SPLINE
SPL {X  -162.820, Y  +621.304, Z    +0.000, E1   +22.259, E3 +549839.256}
SPL {X  -162.820, Y  +618.758, Z    +0.000, E1   +22.239, E3 +549852.407}
SPL {X  -162.820, Y  +616.062, Z    +0.000, E1   +22.275, E3 +549865.828}
SPL {X  -162.820, Y  +613.536, Z    +0.000, E1   +22.242, E3 +549878.949}
SPL {X  -162.820, Y  +611.128, Z    +0.000, E1   +22.252, E3 +549891.120}
SPL {X  -162.820, Y  +608.428, Z    +0.000, E1   +22.255, E3 +549904.904}
SPL {X  -162.820, Y  +605.178, Z    +0.000, E1   +22.267, E3 +549921.436}
SPL {X  -162.820, Y  +602.350, Z    +0.000, E1   +22.224, E3 +549936.053}
SPL {X  -162.820, Y  +599.842, Z    +0.000, E1   +22.298, E3 +549948.204}
SPL {X  -162.820, Y  +597.194, Z    +0.000, E1   +22.253, E3 +549962.125}
SPL {X  -162.820, Y  +594.779, Z    +0.000, E1   +22.284, E3 +549974.029}
SPL {X  -162.820, Y  +592.389, Z    +0.000, E1   +22.245, E3 +549986.646}
SPL {X  -162.820, Y  +589.492, Z    +0.000, E1   +22.304, E3 +550000.830}
SPL {X  -162.820, Y  +587.447, Z    +0.000, E1   +22.279, E3 +550011.359}
SPL {X  -162.820, Y  +585.192, Z    +0.000, E1   +22.298, E3 +550022.769}
SPL {X  -162.820, Y  +582.610, Z    +0.000, E1   +22.234, E3 +550036.393}
SPL {X  -162.820, Y  +580.317, Z    +0.000, E1   +22.300, E3 +550047.447}
SPL {X  -162.820, Y  +578.878, Z    +0.000, E1   +22.272, E3 +550054.956}
SPL {X  -162.820, Y  +576.856, Z    +0.000, E1   +22.233, E3 +550065.715}
SPL {X  -162.820, Y  +574.811, Z    +0.000, E1   +22.236, E3 +550075.978}
SPL {X  -162.820, Y  +572.645, Z    +0.000, E1   +22.246, E3 +550087.074}
SPL {X  -162.820, Y  +569.475, Z    +0.000, E1   +22.269, E3 +550103.080}
SPL {X  -162.820, Y  +565.838, Z    +0.000, E1   +22.271, E3 +550121.675}
SPL {X  -162.820, Y  +562.162, Z    +0.000, E1   +22.252, E3 +550140.492}
SPL {X  -162.820, Y  +558.919, Z    +0.000, E1   +22.286, E3 +550156.655}
SPL {X  -162.820, Y  +556.169, Z    +0.000, E1   +22.295, E3 +550170.484}
SPL {X  -162.820, Y  +553.294, Z    +0.000, E1   +22.266, E3 +550185.482}
SPL {X  -162.820, Y  +550.136, Z    +0.000, E1   +22.258, E3 +550201.595}
SPL {X  -162.820, Y  +546.694, Z    +0.000, E1   +22.290, E3 +550218.917}
SPL {X  -162.820, Y  +543.558, Z    +0.000, E1   +22.285, E3 +550234.780}
SPL {X  -162.820, Y  +541.633, Z    +0.000, E1   +22.257, E3 +550244.708}
SPL {X  -162.820, Y  +539.116, Z    +0.000, E1   +22.302, E3 +550257.319}
SPL {X  -162.820, Y  +536.913, Z    +0.000, E1   +22.192, E3 +550269.243}
SPL {X  -162.820, Y  +534.880, Z    +0.000, E1   +22.252, E3 +550279.197}
SPL {X  -162.820, Y  +532.896, Z    +0.000, E1   +22.234, E3 +550289.357}
SPL {X  -162.820, Y  +531.056, Z    +0.000, E1   +22.251, E3 +550298.639}
SPL {X  -162.820, Y  +528.708, Z    +0.000, E1   +22.319, E3 +550310.021}
SPL {X  -162.820, Y  +525.932, Z    +0.000, E1   +22.258, E3 +550324.777}
SPL {X  -162.820, Y  +522.524, Z    +0.000, E1   +22.326, E3 +550341.501}
SPL {X  -162.820, Y  +519.457, Z    +0.000, E1   +22.481, E3 +550355.630}
SPL {X  -162.820, Y  +506.285, Z    +0.000, E1   +28.538, E3 +550367.088}
SPL {X  -162.820, Y  +504.441, Z    +0.000, E1   +27.574, E3 +550381.430}
SPL {X  -162.820, Y  +503.215, Z    +0.000, E1   +26.369, E3 +550394.937}
SPL {X  -162.820, Y  +502.265, Z    +0.000, E1   +25.287, E3 +550407.419}
SPL {X  -162.820, Y  +501.060, Z    +0.000, E1   +24.081, E3 +550422.160}
SPL {X  -162.820, Y  +500.336, Z    +0.000, E1   +23.110, E3 +550433.299}
SPL {X  -162.820, Y  +499.240, Z    +0.000, E1   +22.316, E3 +550445.610}
SPL {X  -162.820, Y  +498.027, Z    +0.000, E1   +21.516, E3 +550458.518}
SPL {X  -162.820, Y  +495.897, Z    +0.000, E1   +21.662, E3 +550468.438}
SPL {X  -162.820, Y  +493.717, Z    +0.000, E1   +21.704, E3 +550479.544}
SPL {X  -162.820, Y  +491.396, Z    +0.000, E1   +21.707, E3 +550491.668}
SPL {X  -162.820, Y  +488.560, Z    +0.000, E1   +21.695, E3 +550506.778}
SPL {X  -162.820, Y  +485.661, Z    +0.000, E1   +21.712, E3 +550521.663}
SPL {X  -162.820, Y  +483.668, Z    +0.000, E1   +21.664, E3 +550532.491}
SPL {X  -162.820, Y  +481.739, Z    +0.000, E1   +21.704, E3 +550542.204}
SPL {X  -162.820, Y  +479.894, Z    +0.000, E1   +21.695, E3 +550551.992}
SPL {X  -162.820, Y  +477.685, Z    +0.000, E1   +21.656, E3 +550563.929}
SPL {X  -162.820, Y  +475.419, Z    +0.000, E1   +21.711, E3 +550575.282}
SPL {X  -162.820, Y  +473.301, Z    +0.000, E1   +21.712, E3 +550586.379}
SPL {X  -162.820, Y  +470.965, Z    +0.000, E1   +21.700, E3 +550598.724}
SPL {X  -162.820, Y  +469.036, Z    +0.000, E1   +21.695, E3 +550608.768}
SPL {X  -162.820, Y  +467.138, Z    +0.000, E1   +21.678, E3 +550618.939}
SPL {X  -162.820, Y  +465.011, Z    +0.000, E1   +21.692, E3 +550629.922}
SPL {X  -162.820, Y  +462.669, Z    +0.000, E1   +21.752, E3 +550641.702}
SPL {X  -162.820, Y  +460.725, Z    +0.000, E1   +21.689, E3 +550652.315}
SPL {X  -162.820, Y  +458.666, Z    +0.000, E1   +21.695, E3 +550663.127}
SPL {X  -162.820, Y  +456.431, Z    +0.000, E1   +21.708, E3 +550674.656}
SPL {X  -162.820, Y  +454.628, Z    +0.000, E1   +21.674, E3 +550684.374}
SPL {X  -162.820, Y  +452.690, Z    +0.000, E1   +21.773, E3 +550693.648}
SPL {X  -162.820, Y  +450.610, Z    +0.000, E1   +21.698, E3 +550705.247}
SPL {X  -162.820, Y  +448.170, Z    +0.000, E1   +21.667, E3 +550718.268}
SPL {X  -162.820, Y  +446.246, Z    +0.000, E1   +21.696, E3 +550728.086}
SPL {X  -162.820, Y  +443.784, Z    +0.000, E1   +21.713, E3 +550740.872}
SPL {X  -162.820, Y  +441.754, Z    +0.000, E1   +21.708, E3 +550751.424}
SPL {X  -162.820, Y  +439.933, Z    +0.000, E1   +21.690, E3 +550761.188}
SPL {X  -162.820, Y  +437.628, Z    +0.000, E1   +21.678, E3 +550773.376}
SPL {X  -162.820, Y  +435.262, Z    +0.000, E1   +21.727, E3 +550785.311}
SPL {X  -162.820, Y  +433.510, Z    +0.000, E1   +21.692, E3 +550794.725}
SPL {X  -162.820, Y  +431.492, Z    +0.000, E1   +21.686, E3 +550805.421}
SPL {X  -162.820, Y  +429.074, Z    +0.000, E1   +21.710, E3 +550817.873}
SPL {X  -162.820, Y  +427.020, Z    +0.000, E1   +21.674, E3 +550828.874}
SPL {X  -162.820, Y  +425.215, Z    +0.000, E1   +21.693, E3 +550838.177}
SPL {X  -162.820, Y  +422.986, Z    +0.000, E1   +21.685, E3 +550849.988}
SPL {X  -162.820, Y  +420.528, Z    +0.000, E1   +21.706, E3 +550862.638}
SPL {X  -162.820, Y  +418.116, Z    +0.000, E1   +21.761, E3 +550874.785}
SPL {X  -162.820, Y  +416.127, Z    +0.000, E1   +21.715, E3 +550885.490}
SPL {X  -162.820, Y  +414.361, Z    +0.000, E1   +21.613, E3 +550895.678}
SPL {X  -162.820, Y  +411.450, Z    +0.000, E1   +21.710, E3 +550910.251}
SPL {X  -162.820, Y  +408.590, Z    +0.000, E1   +21.735, E3 +550924.877}
SPL {X  -162.820, Y  +406.238, Z    +0.000, E1   +21.697, E3 +550937.526}
SPL {X  -162.820, Y  +404.001, Z    +0.000, E1   +21.723, E3 +550948.955}
SPL {X  -162.820, Y  +402.223, Z    +0.000, E1   +21.697, E3 +550958.440}
SPL {X  -162.820, Y  +400.348, Z    +0.000, E1   +21.713, E3 +550968.166}
SPL {X  -162.820, Y  +398.298, Z    +0.000, E1   +21.721, E3 +550978.782}
SPL {X  -162.820, Y  +396.371, Z    +0.000, E1   +21.713, E3 +550988.964}
SPL {X  -162.820, Y  +394.508, Z    +0.000, E1   +21.616, E3 +550999.519}
SPL {X  -162.820, Y  +392.435, Z    +0.000, E1   +21.681, E3 +551009.873}
SPL {X  -162.820, Y  +389.390, Z    +0.000, E1   +21.742, E3 +551025.479}
SPL {X  -162.820, Y  +386.818, Z    +0.000, E1   +21.679, E3 +551039.238}
SPL {X  -162.820, Y  +384.697, Z    +0.000, E1   +21.693, E3 +551050.308}
SPL {X  -162.820, Y  +382.288, Z    +0.000, E1   +21.742, E3 +551062.432}
SPL {X  -162.820, Y  +380.381, Z    +0.000, E1   +21.655, E3 +551073.157}
SPL {X  -162.808, Y  +378.512, Z    +0.000, E1   +21.736, E3 +551082.209}
SPL {X  -162.776, Y  +376.710, Z    +0.000, E1   +21.698, E3 +551092.008}
SPL {X  -162.707, Y  +374.438, Z    +0.000, E1   +21.688, E3 +551104.012}
SPL {X  -162.607, Y  +372.171, Z    +0.000, E1   +21.692, E3 +551115.812}
SPL {X  -162.494, Y  +370.197, Z    +0.000, E1   +21.655, E3 +551126.438}
SPL {X  -162.349, Y  +368.131, Z    +0.000, E1   +21.624, E3 +551137.556}
SPL {X  -162.161, Y  +365.866, Z    +0.000, E1   +21.642, E3 +551149.241}
SPL {X  -161.927, Y  +363.466, Z    +0.000, E1   +21.730, E3 +551161.013}
SPL {X  -160.290, Y  +351.907, Z    +0.000, E1   +27.562, E3 +551168.591}
SPL {X  -159.725, Y  +348.905, Z    +0.000, E1   +26.136, E3 +551193.826}
ENDSPLINE

SPLINE
SPL {X  -160.871, Y  +355.385, Z    +0.000, E1   +21.841, E3 +551202.669}
SPL {X  -161.833, Y  +362.603, Z    +0.000, E1   +17.021, E3 +551212.700}
ENDSPLINE

SPLINE
SPL {X  -160.786, Y  +354.842, Z    +0.000, E1   +19.274, E3 +551244.855}
ENDSPLINE

SPLINE
SPL {X  -162.485, Y  +370.062, Z    +0.000, E1   +10.606, E3 +551251.233}
SPL {X  -162.818, Y  +379.636, Z    +0.000, E1    +5.115, E3 +551240.582}
SPL {X  -162.820, Y  +386.976, Z    +0.000, E1    +0.144, E3 +551239.681}
SPL {X  -162.820, Y  +391.982, Z    +0.000, E1    -3.443, E3 +551246.446}
SPL {X  -162.820, Y  +399.630, Z    +0.000, E1    -9.426, E3 +551248.954}
SPL {X  -162.820, Y  +408.127, Z    +0.000, E1   -18.417, E3 +551235.242}
SPL {X  -162.820, Y  +420.083, Z    +0.000, E1   -24.325, E3 +551255.718}
SPL {X  -162.820, Y  +428.527, Z    +0.000, E1   -26.988, E3 +551273.010}
SPL {X  -162.820, Y  +431.191, Z    +0.000, E1   -23.548, E3 +551307.863}
SPL {X  -162.820, Y  +432.946, Z    +0.000, E1   -22.795, E3 +551322.266}
SPL {X  -162.820, Y  +434.888, Z    +0.000, E1   -22.823, E3 +551331.673}
SPL {X  -162.820, Y  +436.834, Z    +0.000, E1   -22.779, E3 +551341.633}
SPL {X  -162.820, Y  +438.868, Z    +0.000, E1   -22.837, E3 +551351.287}
SPL {X  -162.820, Y  +441.351, Z    +0.000, E1   -22.805, E3 +551363.862}
SPL {X  -162.820, Y  +443.809, Z    +0.000, E1   -22.804, E3 +551376.028}
SPL {X  -162.820, Y  +446.105, Z    +0.000, E1   -22.815, E3 +551387.270}
SPL {X  -162.820, Y  +447.974, Z    +0.000, E1   -22.856, E3 +551396.173}
SPL {X  -162.820, Y  +449.911, Z    +0.000, E1   -22.774, E3 +551406.448}
SPL {X  -162.820, Y  +451.861, Z    +0.000, E1   -22.750, E3 +551416.295}
SPL {X  -162.820, Y  +454.167, Z    +0.000, E1   -22.842, E3 +551427.025}
SPL {X  -162.820, Y  +456.529, Z    +0.000, E1   -22.855, E3 +551438.553}
SPL {X  -162.820, Y  +458.725, Z    +0.000, E1   -22.793, E3 +551449.958}
SPL {X  -162.820, Y  +461.700, Z    +0.000, E1   -22.822, E3 +551464.580}
SPL {X  -162.820, Y  +464.633, Z    +0.000, E1   -22.813, E3 +551479.077}
SPL {X  -162.820, Y  +466.699, Z    +0.000, E1   -22.824, E3 +551489.123}
SPL {X  -162.820, Y  +468.655, Z    +0.000, E1   -22.858, E3 +551498.567}
SPL {X  -162.820, Y  +470.892, Z    +0.000, E1   -22.837, E3 +551509.805}
SPL {X  -162.820, Y  +472.726, Z    +0.000, E1   -22.777, E3 +551519.344}
SPL {X  -162.820, Y  +475.118, Z    +0.000, E1   -22.777, E3 +551531.316}
SPL {X  -162.820, Y  +478.177, Z    +0.000, E1   -22.834, E3 +551546.008}
SPL {X  -162.820, Y  +481.034, Z    +0.000, E1   -22.831, E3 +551560.146}
SPL {X  -162.820, Y  +483.391, Z    +0.000, E1   -22.793, E3 +551572.082}
SPL {X  -162.820, Y  +486.307, Z    +0.000, E1   -22.833, E3 +551586.336}
SPL {X  -162.820, Y  +488.828, Z    +0.000, E1   -22.793, E3 +551598.979}
SPL {X  -162.820, Y  +491.768, Z    +0.000, E1   -22.852, E3 +551613.276}
SPL {X  -162.820, Y  +495.526, Z    +0.000, E1   -22.833, E3 +551632.047}
SPL {X  -162.820, Y  +499.330, Z    +0.000, E1   -22.841, E3 +551650.828}
SPL {X  -162.820, Y  +503.049, Z    +0.000, E1   -22.823, E3 +551669.377}
SPL {X  -162.820, Y  +506.908, Z    +0.000, E1   -22.877, E3 +551688.047}
SPL {X  -162.820, Y  +510.068, Z    +0.000, E1   -22.761, E3 +551704.519}
SPL {X  -162.820, Y  +512.359, Z    +0.000, E1   -22.823, E3 +551715.250}
SPL {X  -162.820, Y  +513.873, Z    +0.000, E1   -22.800, E3 +551722.937}
SPL {X  -162.820, Y  +516.100, Z    +0.000, E1   -22.809, E3 +551734.014}
SPL {X  -162.820, Y  +518.662, Z    +0.000, E1   -22.847, E3 +551746.312}
SPL {X  -162.820, Y  +520.641, Z    +0.000, E1   -22.790, E3 +551756.553}
SPL {X  -162.820, Y  +523.535, Z    +0.000, E1   -22.857, E3 +551770.522}
SPL {X  -162.820, Y  +526.661, Z    +0.000, E1   -22.801, E3 +551786.346}
SPL {X  -162.820, Y  +528.725, Z    +0.000, E1   -22.770, E3 +551796.715}
SPL {X  -162.820, Y  +530.303, Z    +0.000, E1   -22.798, E3 +551804.335}
SPL {X  -162.820, Y  +532.614, Z    +0.000, E1   -22.828, E3 +551815.603}
SPL {X  -162.820, Y  +534.838, Z    +0.000, E1   -22.864, E3 +551826.232}
SPL {X  -162.820, Y  +536.882, Z    +0.000, E1   -22.782, E3 +551837.087}
SPL {X  -162.820, Y  +539.194, Z    +0.000, E1   -22.826, E3 +551848.135}
SPL {X  -162.820, Y  +541.555, Z    +0.000, E1   -22.817, E3 +551859.950}
SPL {X  -162.820, Y  +543.728, Z    +0.000, E1   -22.799, E3 +551870.807}
SPL {X  -162.820, Y  +545.925, Z    +0.000, E1   -22.803, E3 +551881.677}
SPL {X  -162.820, Y  +549.071, Z    +0.000, E1   -22.836, E3 +551897.205}
SPL {X  -162.820, Y  +553.089, Z    +0.000, E1   -22.838, E3 +551917.105}
SPL {X  -162.820, Y  +556.430, Z    +0.000, E1   -22.821, E3 +551933.606}
SPL {X  -162.820, Y  +558.974, Z    +0.000, E1   -22.806, E3 +551946.306}
SPL {X  -162.820, Y  +562.171, Z    +0.000, E1   -22.845, E3 +551962.004}
SPL {X  -162.820, Y  +565.170, Z    +0.000, E1   -22.801, E3 +551977.017}
SPL {X  -162.820, Y  +567.308, Z    +0.000, E1   -22.750, E3 +551988.033}
SPL {X  -162.820, Y  +570.378, Z    +0.000, E1   -22.843, E3 +552002.657}
SPL {X  -162.820, Y  +573.634, Z    +0.000, E1   -22.827, E3 +552018.801}
SPL {X  -162.820, Y  +576.228, Z    +0.000, E1   -22.814, E3 +552031.697}
SPL {X  -162.820, Y  +578.553, Z    +0.000, E1   -22.801, E3 +552043.313}
SPL {X  -162.820, Y  +581.064, Z    +0.000, E1   -22.823, E3 +552055.597}
SPL {X  -162.820, Y  +583.435, Z    +0.000, E1   -22.808, E3 +552067.419}
SPL {X  -162.820, Y  +585.410, Z    +0.000, E1   -22.764, E3 +552077.555}
SPL {X  -162.820, Y  +587.676, Z    +0.000, E1   -22.853, E3 +552088.069}
SPL {X  -162.820, Y  +590.707, Z    +0.000, E1   -22.855, E3 +552103.220}
SPL {X  -162.820, Y  +593.650, Z    +0.000, E1   -22.810, E3 +552117.980}
SPL {X  -162.820, Y  +595.830, Z    +0.000, E1   -22.828, E3 +552128.596}
SPL {X  -162.820, Y  +598.094, Z    +0.000, E1   -22.843, E3 +552139.709}
SPL {X  -162.820, Y  +600.420, Z    +0.000, E1   -22.826, E3 +552151.340}
SPL {X  -162.820, Y  +602.573, Z    +0.000, E1   -22.830, E3 +552161.925}
SPL {X  -162.820, Y  +604.828, Z    +0.000, E1   -22.784, E3 +552173.564}
SPL {X  -162.820, Y  +608.133, Z    +0.000, E1   -22.831, E3 +552189.682}
SPL {X  -162.820, Y  +611.103, Z    +0.000, E1   -22.785, E3 +552204.607}
SPL {X  -162.820, Y  +613.294, Z    +0.000, E1   -22.780, E3 +552215.480}
SPL {X  -162.820, Y  +615.356, Z    +0.000, E1   -22.799, E3 +552225.538}
SPL {X  -162.820, Y  +617.439, Z    +0.000, E1   -22.808, E3 +552235.796}
SPL {X  -162.820, Y  +619.665, Z    +0.000, E1   -22.817, E3 +552246.764}
SPL {X  -162.820, Y  +621.733, Z    +0.000, E1   -22.759, E3 +552257.488}
SPL {X  -162.820, Y  +624.076, Z    +0.000, E1   -22.774, E3 +552268.993}
SPL {X  -162.820, Y  +627.244, Z    +0.000, E1   -22.803, E3 +552284.675}
SPL {X  -162.820, Y  +630.349, Z    +0.000, E1   -22.766, E3 +552300.207}
SPL {X  -162.820, Y  +632.572, Z    +0.000, E1   -22.785, E3 +552311.014}
SPL {X  -162.820, Y  +634.507, Z    +0.000, E1   -22.784, E3 +552320.653}
SPL {X  -162.820, Y  +636.863, Z    +0.000, E1   -22.760, E3 +552332.575}
SPL {X  -162.820, Y  +640.111, Z    +0.000, E1   -22.809, E3 +552348.458}
SPL {X  -162.820, Y  +643.449, Z    +0.000, E1   -22.796, E3 +552364.975}
SPL {X  -162.820, Y  +645.630, Z    +0.000, E1   -22.795, E3 +552375.671}
SPL {X  -162.820, Y  +647.561, Z    +0.000, E1   -22.705, E3 +552386.122}
SPL {X  -162.820, Y  +651.051, Z    +0.000, E1   -22.833, E3 +552402.542}
SPL {X  -162.820, Y  +653.898, Z    +0.000, E1   -22.796, E3 +552416.727}
SPL {X  -162.820, Y  +656.161, Z    +0.000, E1   -22.812, E3 +552427.849}
SPL {X  -162.820, Y  +658.384, Z    +0.000, E1   -22.822, E3 +552438.715}
SPL {X  -162.820, Y  +660.215, Z    +0.000, E1   -22.649, E3 +552449.306}
SPL {X  -162.820, Y  +662.823, Z    +0.000, E1   -22.799, E3 +552461.014}
SPL {X  -162.820, Y  +665.862, Z    +0.000, E1   -22.864, E3 +552475.713}
SPL {X  -162.820, Y  +668.960, Z    +0.000, E1   -22.773, E3 +552491.664}
SPL {X  -162.820, Y  +672.333, Z    +0.000, E1   -22.837, E3 +552508.000}
SPL {X  -162.812, Y  +675.071, Z    +0.000, E1   -22.742, E3 +552522.145}
SPL {X  -162.773, Y  +677.428, Z    +0.000, E1   -22.762, E3 +552533.743}
SPL {X  -162.691, Y  +679.987, Z    +0.000, E1   -22.794, E3 +552546.156}
SPL {X  -162.604, Y  +681.880, Z    +0.000, E1   -22.691, E3 +552556.317}
SPL {X  -162.458, Y  +684.346, Z    +0.000, E1   -22.764, E3 +552568.110}
SPL {X  -162.296, Y  +686.547, Z    +0.000, E1   -22.660, E3 +552579.727}
SPL {X  -162.090, Y  +688.902, Z    +0.000, E1   -22.700, E3 +552591.235}
SPL {X  -161.474, Y  +694.390, Z    +0.000, E1   -24.298, E3 +552604.590}
SPL {X  -158.730, Y  +709.763, Z    +0.000, E1   -31.225, E3 +552615.929}
ENDSPLINE

SPLINE
SPL {X  -160.932, Y  +698.225, Z    +0.000, E1   -21.712, E3 +552647.038}
SPL {X  -161.917, Y  +690.622, Z    +0.000, E1   -16.445, E3 +552660.639}
ENDSPLINE

SPLINE
SPL {X  -161.349, Y  +695.340, Z    +0.000, E1   -18.625, E3 +552668.258}
ENDSPLINE

SPLINE
SPL {X  -162.534, Y  +683.153, Z    +0.000, E1   -10.475, E3 +552689.388}
SPL {X  -162.820, Y  +667.630, Z    +0.000, E1    -0.882, E3 +552683.365}
SPL {X  -162.820, Y  +661.883, Z    +0.000, E1    +3.373, E3 +552688.808}
SPL {X  -162.820, Y  +653.808, Z    +0.000, E1    +9.891, E3 +552686.499}
SPL {X  -162.820, Y  +632.548, Z    +0.000, E1   +27.446, E3 +552683.036}
ENDSPLINE

SPLINE
SPL {X  -162.820, Y  +638.080, Z    +0.000, E1   +18.858, E3 +552710.784}
ENDSPLINE

SPLINE
SPL {X  -162.820, Y  +623.278, Z    +0.000, E1   +28.723, E3 +552712.355}
SPL {X  -162.820, Y  +618.658, Z    +0.000, E1   +26.841, E3 +552740.964}
ENDSPLINE

SPLINE
SPL {X  -162.820, Y  +623.685, Z    +0.000, E1   +22.346, E3 +552753.271}
ENDSPLINE

SPLINE
SPL {X  -162.820, Y  +621.304, Z    +0.000, E1   +22.259, E3 +552766.086}
SPL {X  -162.820, Y  +618.758, Z    +0.000, E1   +22.239, E3 +552779.237}
SPL {X  -162.820, Y  +616.062, Z    +0.000, E1   +22.275, E3 +552792.657}
SPL {X  -162.820, Y  +613.536, Z    +0.000, E1   +22.242, E3 +552805.779}
SPL {X  -162.820, Y  +610.461, Z    +0.000, E1   +22.264, E3 +552821.410}
SPL {X  -162.820, Y  +607.796, Z    +0.000, E1   +22.261, E3 +552834.781}
SPL {X  -162.820, Y  +605.178, Z    +0.000, E1   +22.267, E3 +552848.265}
SPL {X  -162.820, Y  +602.350, Z    +0.000, E1   +22.224, E3 +552862.882}
SPL {X  -162.820, Y  +599.842, Z    +0.000, E1   +22.298, E3 +552875.034}
SPL {X  -162.820, Y  +597.194, Z    +0.000, E1   +22.253, E3 +552888.955}
SPL {X  -162.820, Y  +594.779, Z    +0.000, E1   +22.284, E3 +552900.859}
SPL {X  -162.820, Y  +592.389, Z    +0.000, E1   +22.245, E3 +552913.475}
SPL {X  -162.820, Y  +589.492, Z    +0.000, E1   +22.304, E3 +552927.659}
SPL {X  -162.820, Y  +587.447, Z    +0.000, E1   +22.279, E3 +552938.188}
SPL {X  -162.820, Y  +585.192, Z    +0.000, E1   +22.298, E3 +552949.599}
SPL {X  -162.820, Y  +582.610, Z    +0.000, E1   +22.234, E3 +552963.222}
SPL {X  -162.820, Y  +580.317, Z    +0.000, E1   +22.300, E3 +552974.276}
SPL {X  -162.820, Y  +578.878, Z    +0.000, E1   +22.272, E3 +552981.785}
SPL {X  -162.820, Y  +576.856, Z    +0.000, E1   +22.233, E3 +552992.544}
SPL {X  -162.820, Y  +574.811, Z    +0.000, E1   +22.236, E3 +553002.807}
SPL {X  -162.820, Y  +572.645, Z    +0.000, E1   +22.246, E3 +553013.903}
SPL {X  -162.820, Y  +570.282, Z    +0.000, E1   +22.231, E3 +553025.953}
SPL {X  -162.820, Y  +567.961, Z    +0.000, E1   +22.247, E3 +553037.743}
SPL {X  -162.820, Y  +564.506, Z    +0.000, E1   +22.298, E3 +553055.057}
SPL {X  -162.820, Y  +561.620, Z    +0.000, E1   +22.191, E3 +553070.438}
SPL {X  -162.820, Y  +559.515, Z    +0.000, E1   +22.273, E3 +553080.440}
SPL {X  -162.820, Y  +556.723, Z    +0.000, E1   +22.309, E3 +553094.523}
SPL {X  -162.820, Y  +554.378, Z    +0.000, E1   +22.288, E3 +553106.369}
SPL {X  -162.820, Y  +552.787, Z    +0.000, E1   +22.213, E3 +553115.191}
SPL {X  -162.820, Y  +550.871, Z    +0.000, E1   +22.229, E3 +553124.785}
SPL {X  -162.820, Y  +548.168, Z    +0.000, E1   +22.298, E3 +553138.121}
SPL {X  -162.820, Y  +545.860, Z    +0.000, E1   +22.216, E3 +553150.379}
SPL {X  -162.820, Y  +543.558, Z    +0.000, E1   +22.285, E3 +553161.609}
SPL {X  -162.820, Y  +541.633, Z    +0.000, E1   +22.257, E3 +553171.538}
SPL {X  -162.820, Y  +539.116, Z    +0.000, E1   +22.302, E3 +553184.148}
SPL {X  -162.820, Y  +535.523, Z    +0.000, E1   +22.266, E3 +553202.810}
SPL {X  -162.820, Y  +531.757, Z    +0.000, E1   +22.276, E3 +553221.864}
SPL {X  -162.820, Y  +527.980, Z    +0.000, E1   +22.326, E3 +553240.695}
SPL {X  -162.820, Y  +524.599, Z    +0.000, E1   +22.287, E3 +553258.093}
SPL {X  -162.820, Y  +522.011, Z    +0.000, E1   +22.282, E3 +553271.170}
SPL {X  -162.820, Y  +519.457, Z    +0.000, E1   +22.481, E3 +553282.459}
SPL {X  -162.820, Y  +506.285, Z    +0.000, E1   +28.538, E3 +553293.917}
SPL {X  -162.820, Y  +504.441, Z    +0.000, E1   +27.574, E3 +553308.259}
SPL {X  -162.820, Y  +502.813, Z    +0.000, E1   +26.013, E3 +553326.457}
SPL {X  -162.820, Y  +502.016, Z    +0.000, E1   +24.802, E3 +553338.799}
SPL {X  -162.820, Y  +501.060, Z    +0.000, E1   +24.081, E3 +553348.989}
SPL {X  -162.820, Y  +500.336, Z    +0.000, E1   +23.110, E3 +553360.129}
SPL {X  -162.820, Y  +499.240, Z    +0.000, E1   +22.316, E3 +553372.440}
SPL {X  -162.820, Y  +498.027, Z    +0.000, E1   +21.516, E3 +553385.347}
SPL {X  -162.820, Y  +495.897, Z    +0.000, E1   +21.662, E3 +553395.267}
SPL {X  -162.820, Y  +493.717, Z    +0.000, E1   +21.704, E3 +553406.374}
SPL {X  -162.820, Y  +491.396, Z    +0.000, E1   +21.707, E3 +553418.498}
SPL {X  -162.820, Y  +488.560, Z    +0.000, E1   +21.695, E3 +553433.607}
SPL {X  -162.820, Y  +485.661, Z    +0.000, E1   +21.712, E3 +553448.492}
SPL {X  -162.820, Y  +483.668, Z    +0.000, E1   +21.664, E3 +553459.320}
SPL {X  -162.820, Y  +481.739, Z    +0.000, E1   +21.704, E3 +553469.034}
SPL {X  -162.820, Y  +479.894, Z    +0.000, E1   +21.695, E3 +553478.821}
SPL {X  -162.820, Y  +477.685, Z    +0.000, E1   +21.656, E3 +553490.759}
SPL {X  -162.820, Y  +475.419, Z    +0.000, E1   +21.711, E3 +553502.111}
SPL {X  -162.820, Y  +473.301, Z    +0.000, E1   +21.712, E3 +553513.208}
SPL {X  -162.820, Y  +470.965, Z    +0.000, E1   +21.700, E3 +553525.553}
SPL {X  -162.820, Y  +469.036, Z    +0.000, E1   +21.695, E3 +553535.597}
SPL {X  -162.820, Y  +467.138, Z    +0.000, E1   +21.678, E3 +553545.769}
SPL {X  -162.820, Y  +465.011, Z    +0.000, E1   +21.692, E3 +553556.751}
SPL {X  -162.820, Y  +462.669, Z    +0.000, E1   +21.752, E3 +553568.532}
SPL {X  -162.820, Y  +460.725, Z    +0.000, E1   +21.689, E3 +553579.145}
SPL {X  -162.820, Y  +458.666, Z    +0.000, E1   +21.695, E3 +553589.957}
SPL {X  -162.820, Y  +456.431, Z    +0.000, E1   +21.708, E3 +553601.485}
SPL {X  -162.820, Y  +453.609, Z    +0.000, E1   +21.757, E3 +553616.019}
SPL {X  -162.820, Y  +450.610, Z    +0.000, E1   +21.698, E3 +553632.076}
SPL {X  -162.820, Y  +448.170, Z    +0.000, E1   +21.667, E3 +553645.097}
SPL {X  -162.820, Y  +446.246, Z    +0.000, E1   +21.696, E3 +553654.915}
SPL {X  -162.820, Y  +443.784, Z    +0.000, E1   +21.713, E3 +553667.701}
SPL {X  -162.820, Y  +440.567, Z    +0.000, E1   +21.731, E3 +553684.541}
SPL {X  -162.820, Y  +437.628, Z    +0.000, E1   +21.678, E3 +553700.205}
SPL {X  -162.820, Y  +434.473, Z    +0.000, E1   +21.747, E3 +553716.301}
SPL {X  -162.820, Y  +431.492, Z    +0.000, E1   +21.686, E3 +553732.250}
SPL {X  -162.820, Y  +429.074, Z    +0.000, E1   +21.710, E3 +553744.702}
SPL {X  -162.820, Y  +426.023, Z    +0.000, E1   +21.718, E3 +553760.770}
SPL {X  -162.820, Y  +422.986, Z    +0.000, E1   +21.685, E3 +553776.817}
SPL {X  -162.820, Y  +420.528, Z    +0.000, E1   +21.706, E3 +553789.467}
SPL {X  -162.820, Y  +418.116, Z    +0.000, E1   +21.761, E3 +553801.614}
SPL {X  -162.820, Y  +416.127, Z    +0.000, E1   +21.715, E3 +553812.320}
SPL {X  -162.820, Y  +414.361, Z    +0.000, E1   +21.613, E3 +553822.507}
SPL {X  -162.820, Y  +411.450, Z    +0.000, E1   +21.710, E3 +553837.080}
SPL {X  -162.820, Y  +408.590, Z    +0.000, E1   +21.735, E3 +553851.706}
SPL {X  -162.820, Y  +406.238, Z    +0.000, E1   +21.697, E3 +553864.355}
SPL {X  -162.820, Y  +403.166, Z    +0.000, E1   +21.746, E3 +553880.161}
SPL {X  -162.820, Y  +400.348, Z    +0.000, E1   +21.713, E3 +553894.995}
SPL {X  -162.820, Y  +398.298, Z    +0.000, E1   +21.721, E3 +553905.611}
SPL {X  -162.820, Y  +396.371, Z    +0.000, E1   +21.713, E3 +553915.793}
SPL {X  -162.820, Y  +394.508, Z    +0.000, E1   +21.616, E3 +553926.348}
SPL {X  -162.820, Y  +391.777, Z    +0.000, E1   +21.714, E3 +553940.008}
SPL {X  -162.820, Y  +388.822, Z    +0.000, E1   +21.717, E3 +553955.327}
SPL {X  -162.820, Y  +386.818, Z    +0.000, E1   +21.679, E3 +553966.067}
SPL {X  -162.820, Y  +384.697, Z    +0.000, E1   +21.693, E3 +553977.138}
SPL {X  -162.820, Y  +382.288, Z    +0.000, E1   +21.742, E3 +553989.261}
SPL {X  -162.817, Y  +379.520, Z    +0.000, E1   +21.723, E3 +554004.099}
SPL {X  -162.776, Y  +376.710, Z    +0.000, E1   +21.698, E3 +554018.838}
SPL {X  -162.707, Y  +374.438, Z    +0.000, E1   +21.688, E3 +554030.842}
SPL {X  -162.607, Y  +372.171, Z    +0.000, E1   +21.692, E3 +554042.641}
SPL {X  -162.494, Y  +370.197, Z    +0.000, E1   +21.655, E3 +554053.268}
SPL {X  -162.349, Y  +368.131, Z    +0.000, E1   +21.624, E3 +554064.386}
SPL {X  -162.161, Y  +365.866, Z    +0.000, E1   +21.642, E3 +554076.071}
SPL {X  -161.651, Y  +361.024, Z    +0.000, E1   +22.970, E3 +554089.494}
SPL {X  -160.281, Y  +351.857, Z    +0.000, E1   +24.243, E3 +554124.833}
ENDSPLINE

SPLINE
SPL {X  -161.833, Y  +362.603, Z    +0.000, E1   +17.021, E3 +554139.529}
ENDSPLINE

SPLINE
SPL {X  -160.786, Y  +354.842, Z    +0.000, E1   +19.274, E3 +554171.685}
ENDSPLINE

SPLINE
SPL {X  -162.485, Y  +370.062, Z    +0.000, E1   +10.606, E3 +554178.063}
SPL {X  -162.820, Y  +381.311, Z    +0.000, E1    +4.054, E3 +554168.418}
SPL {X  -162.820, Y  +389.994, Z    +0.000, E1    -2.149, E3 +554162.830}
SPL {X  -162.820, Y  +391.982, Z    +0.000, E1    -3.443, E3 +554173.275}
SPL {X  -162.820, Y  +399.630, Z    +0.000, E1    -9.426, E3 +554175.783}
SPL {X  -162.820, Y  +408.127, Z    +0.000, E1   -18.417, E3 +554162.071}
SPL {X  -162.820, Y  +420.083, Z    +0.000, E1   -24.325, E3 +554182.547}
SPL {X  -162.820, Y  +428.527, Z    +0.000, E1   -26.988, E3 +554199.839}
SPL {X  -162.820, Y  +431.336, Z    +0.000, E1   -24.162, E3 +554230.049}
SPL {X  -162.820, Y  +432.048, Z    +0.000, E1   -22.832, E3 +554244.553}
SPL {X  -162.820, Y  +434.888, Z    +0.000, E1   -22.823, E3 +554258.502}
SPL {X  -162.820, Y  +436.834, Z    +0.000, E1   -22.779, E3 +554268.462}
SPL {X  -162.820, Y  +438.868, Z    +0.000, E1   -22.837, E3 +554278.116}
SPL {X  -162.820, Y  +441.351, Z    +0.000, E1   -22.805, E3 +554290.691}
SPL {X  -162.820, Y  +443.809, Z    +0.000, E1   -22.804, E3 +554302.857}
SPL {X  -162.820, Y  +447.077, Z    +0.000, E1   -22.869, E3 +554318.668}
SPL {X  -162.820, Y  +449.911, Z    +0.000, E1   -22.774, E3 +554333.277}
SPL {X  -162.820, Y  +451.861, Z    +0.000, E1   -22.750, E3 +554343.125}
SPL {X  -162.820, Y  +454.167, Z    +0.000, E1   -22.842, E3 +554353.854}
SPL {X  -162.820, Y  +456.529, Z    +0.000, E1   -22.855, E3 +554365.383}
SPL {X  -162.820, Y  +458.725, Z    +0.000, E1   -22.793, E3 +554376.787}
SPL {X  -162.820, Y  +460.754, Z    +0.000, E1   -22.806, E3 +554386.660}
SPL {X  -162.820, Y  +462.409, Z    +0.000, E1   -22.783, E3 +554395.077}
SPL {X  -162.820, Y  +464.633, Z    +0.000, E1   -22.813, E3 +554405.906}
SPL {X  -162.820, Y  +467.913, Z    +0.000, E1   -22.879, E3 +554421.745}
SPL {X  -162.820, Y  +470.892, Z    +0.000, E1   -22.837, E3 +554436.635}
SPL {X  -162.820, Y  +472.726, Z    +0.000, E1   -22.777, E3 +554446.173}
SPL {X  -162.820, Y  +475.118, Z    +0.000, E1   -22.777, E3 +554458.145}
SPL {X  -162.820, Y  +477.389, Z    +0.000, E1   -22.803, E3 +554469.062}
SPL {X  -162.820, Y  +478.914, Z    +0.000, E1   -22.821, E3 +554476.453}
SPL {X  -162.820, Y  +481.034, Z    +0.000, E1   -22.831, E3 +554486.975}
SPL {X  -162.820, Y  +484.256, Z    +0.000, E1   -22.840, E3 +554502.994}
SPL {X  -162.820, Y  +487.952, Z    +0.000, E1   -22.824, E3 +554521.424}
SPL {X  -162.820, Y  +491.768, Z    +0.000, E1   -22.852, E3 +554540.105}
SPL {X  -162.820, Y  +495.526, Z    +0.000, E1   -22.833, E3 +554558.876}
SPL {X  -162.820, Y  +499.330, Z    +0.000, E1   -22.841, E3 +554577.657}
SPL {X  -162.820, Y  +503.049, Z    +0.000, E1   -22.823, E3 +554596.207}
SPL {X  -162.820, Y  +506.908, Z    +0.000, E1   -22.877, E3 +554614.877}
SPL {X  -162.820, Y  +510.068, Z    +0.000, E1   -22.761, E3 +554631.348}
SPL {X  -162.820, Y  +512.359, Z    +0.000, E1   -22.823, E3 +554642.080}
SPL {X  -162.820, Y  +513.873, Z    +0.000, E1   -22.800, E3 +554649.766}
SPL {X  -162.820, Y  +516.100, Z    +0.000, E1   -22.809, E3 +554660.843}
SPL {X  -162.820, Y  +518.662, Z    +0.000, E1   -22.847, E3 +554673.141}
SPL {X  -162.820, Y  +520.641, Z    +0.000, E1   -22.790, E3 +554683.382}
SPL {X  -162.820, Y  +523.535, Z    +0.000, E1   -22.857, E3 +554697.351}
SPL {X  -162.820, Y  +526.661, Z    +0.000, E1   -22.801, E3 +554713.175}
SPL {X  -162.820, Y  +528.725, Z    +0.000, E1   -22.770, E3 +554723.545}
SPL {X  -162.820, Y  +530.303, Z    +0.000, E1   -22.798, E3 +554731.164}
SPL {X  -162.820, Y  +532.614, Z    +0.000, E1   -22.828, E3 +554742.432}
SPL {X  -162.820, Y  +534.838, Z    +0.000, E1   -22.864, E3 +554753.061}
SPL {X  -162.820, Y  +536.882, Z    +0.000, E1   -22.782, E3 +554763.916}
SPL {X  -162.820, Y  +539.194, Z    +0.000, E1   -22.826, E3 +554774.965}
SPL {X  -162.820, Y  +541.555, Z    +0.000, E1   -22.817, E3 +554786.779}
SPL {X  -162.820, Y  +543.728, Z    +0.000, E1   -22.799, E3 +554797.637}
SPL {X  -162.820, Y  +545.925, Z    +0.000, E1   -22.803, E3 +554808.506}
SPL {X  -162.820, Y  +548.328, Z    +0.000, E1   -22.796, E3 +554820.502}
SPL {X  -162.820, Y  +551.027, Z    +0.000, E1   -22.819, E3 +554833.695}
SPL {X  -162.820, Y  +553.721, Z    +0.000, E1   -22.807, E3 +554847.139}
SPL {X  -162.820, Y  +556.430, Z    +0.000, E1   -22.821, E3 +554860.435}
SPL {X  -162.820, Y  +559.675, Z    +0.000, E1   -22.837, E3 +554876.515}
SPL {X  -162.820, Y  +562.799, Z    +0.000, E1   -22.814, E3 +554892.021}
SPL {X  -162.820, Y  +565.170, Z    +0.000, E1   -22.801, E3 +554903.846}
SPL {X  -162.820, Y  +568.020, Z    +0.000, E1   -22.787, E3 +554918.233}
SPL {X  -162.820, Y  +570.992, Z    +0.000, E1   -22.834, E3 +554932.452}
SPL {X  -162.820, Y  +572.901, Z    +0.000, E1   -22.775, E3 +554942.321}
SPL {X  -162.820, Y  +575.638, Z    +0.000, E1   -22.855, E3 +554955.430}
SPL {X  -162.820, Y  +578.553, Z    +0.000, E1   -22.801, E3 +554970.142}
SPL {X  -162.820, Y  +581.064, Z    +0.000, E1   -22.823, E3 +554982.427}
SPL {X  -162.820, Y  +583.435, Z    +0.000, E1   -22.808, E3 +554994.248}
SPL {X  -162.820, Y  +585.410, Z    +0.000, E1   -22.764, E3 +555004.384}
SPL {X  -162.820, Y  +587.676, Z    +0.000, E1   -22.853, E3 +555014.899}
SPL {X  -162.820, Y  +589.682, Z    +0.000, E1   -22.776, E3 +555025.429}
SPL {X  -162.820, Y  +591.720, Z    +0.000, E1   -22.868, E3 +555034.739}
SPL {X  -162.820, Y  +593.650, Z    +0.000, E1   -22.810, E3 +555044.809}
SPL {X  -162.820, Y  +595.830, Z    +0.000, E1   -22.828, E3 +555055.425}
SPL {X  -162.820, Y  +598.094, Z    +0.000, E1   -22.843, E3 +555066.538}
SPL {X  -162.820, Y  +600.420, Z    +0.000, E1   -22.826, E3 +555078.169}
SPL {X  -162.820, Y  +602.573, Z    +0.000, E1   -22.830, E3 +555088.755}
SPL {X  -162.820, Y  +604.828, Z    +0.000, E1   -22.784, E3 +555100.393}
SPL {X  -162.820, Y  +607.142, Z    +0.000, E1   -22.808, E3 +555111.574}
SPL {X  -162.820, Y  +608.890, Z    +0.000, E1   -22.790, E3 +555120.398}
SPL {X  -162.820, Y  +611.103, Z    +0.000, E1   -22.785, E3 +555131.437}
SPL {X  -162.820, Y  +613.294, Z    +0.000, E1   -22.780, E3 +555142.310}
SPL {X  -162.820, Y  +615.356, Z    +0.000, E1   -22.799, E3 +555152.367}
SPL {X  -162.820, Y  +617.439, Z    +0.000, E1   -22.808, E3 +555162.625}
SPL {X  -162.820, Y  +619.665, Z    +0.000, E1   -22.817, E3 +555173.593}
SPL {X  -162.820, Y  +621.733, Z    +0.000, E1   -22.759, E3 +555184.317}
SPL {X  -162.820, Y  +624.076, Z    +0.000, E1   -22.774, E3 +555195.822}
SPL {X  -162.820, Y  +626.527, Z    +0.000, E1   -22.768, E3 +555208.065}
SPL {X  -162.820, Y  +629.758, Z    +0.000, E1   -22.800, E3 +555223.994}
SPL {X  -162.820, Y  +632.572, Z    +0.000, E1   -22.785, E3 +555237.843}
SPL {X  -162.820, Y  +634.507, Z    +0.000, E1   -22.784, E3 +555247.482}
SPL {X  -162.820, Y  +636.863, Z    +0.000, E1   -22.760, E3 +555259.404}
SPL {X  -162.820, Y  +639.254, Z    +0.000, E1   -22.767, E3 +555271.187}
SPL {X  -162.820, Y  +641.195, Z    +0.000, E1   -22.782, E3 +555280.635}
SPL {X  -162.820, Y  +643.449, Z    +0.000, E1   -22.796, E3 +555291.805}
SPL {X  -162.820, Y  +645.630, Z    +0.000, E1   -22.795, E3 +555302.501}
SPL {X  -162.820, Y  +647.561, Z    +0.000, E1   -22.705, E3 +555312.951}
SPL {X  -162.820, Y  +651.051, Z    +0.000, E1   -22.833, E3 +555329.371}
SPL {X  -162.820, Y  +653.898, Z    +0.000, E1   -22.796, E3 +555343.557}
SPL {X  -162.820, Y  +656.161, Z    +0.000, E1   -22.812, E3 +555354.678}
SPL {X  -162.820, Y  +658.384, Z    +0.000, E1   -22.822, E3 +555365.544}
SPL {X  -162.820, Y  +660.215, Z    +0.000, E1   -22.649, E3 +555376.135}
SPL {X  -162.820, Y  +662.823, Z    +0.000, E1   -22.799, E3 +555387.843}
SPL {X  -162.820, Y  +665.112, Z    +0.000, E1   -22.835, E3 +555398.897}
SPL {X  -162.820, Y  +667.016, Z    +0.000, E1   -22.823, E3 +555408.326}
SPL {X  -162.820, Y  +668.960, Z    +0.000, E1   -22.773, E3 +555418.493}
SPL {X  -162.820, Y  +671.605, Z    +0.000, E1   -22.777, E3 +555431.567}
SPL {X  -162.817, Y  +674.515, Z    +0.000, E1   -22.816, E3 +555445.764}
SPL {X  -162.773, Y  +677.428, Z    +0.000, E1   -22.762, E3 +555460.572}
SPL {X  -162.691, Y  +679.987, Z    +0.000, E1   -22.794, E3 +555472.985}
SPL {X  -162.604, Y  +681.880, Z    +0.000, E1   -22.691, E3 +555483.146}
SPL {X  -162.458, Y  +684.346, Z    +0.000, E1   -22.764, E3 +555494.940}
SPL {X  -162.229, Y  +687.364, Z    +0.000, E1   -22.685, E3 +555510.559}
SPL {X  -161.938, Y  +690.422, Z    +0.000, E1   -22.769, E3 +555524.966}
SPL {X  -161.065, Y  +697.344, Z    +0.000, E1   -25.698, E3 +555534.085}
SPL {X  -158.553, Y  +710.529, Z    +0.000, E1   -30.890, E3 +555547.982}
ENDSPLINE

SPLINE
SPL {X  -161.215, Y  +696.305, Z    +0.000, E1   -20.575, E3 +555574.562}
SPL {X  -161.691, Y  +692.643, Z    +0.000, E1   -17.369, E3 +555590.751}
SPL {X  -162.534, Y  +683.153, Z    +0.000, E1   -10.475, E3 +555616.218}
SPL {X  -162.820, Y  +670.105, Z    +0.000, E1    -2.484, E3 +555608.864}
SPL {X  -162.820, Y  +665.819, Z    +0.000, E1    +0.492, E3 +555611.161}
SPL {X  -162.820, Y  +661.883, Z    +0.000, E1    +3.373, E3 +555615.637}
SPL {X  -162.820, Y  +655.163, Z    +0.000, E1    +8.702, E3 +555615.236}
SPL {X  -162.820, Y  +634.515, Z    +0.000, E1   +26.439, E3 +555607.649}
ENDSPLINE

SPLINE
SPL {X  -162.820, Y  +638.080, Z    +0.000, E1   +18.858, E3 +555637.614}
ENDSPLINE

SPLINE
SPL {X  -162.820, Y  +623.278, Z    +0.000, E1   +28.723, E3 +555639.184}
SPL {X  -162.820, Y  +618.658, Z    +0.000, E1   +26.841, E3 +555667.793}
ENDSPLINE

SPLINE
SPL {X  -162.820, Y  +623.685, Z    +0.000, E1   +22.346, E3 +555680.100}
ENDSPLINE

SPLINE
SPL {X  -162.820, Y  +621.304, Z    +0.000, E1   +22.259, E3 +555692.915}
SPL {X  -162.820, Y  +618.758, Z    +0.000, E1   +22.239, E3 +555706.066}
SPL {X  -162.820, Y  +616.062, Z    +0.000, E1   +22.275, E3 +555719.486}
SPL {X  -162.820, Y  +613.536, Z    +0.000, E1   +22.242, E3 +555732.608}
SPL {X  -162.820, Y  +611.128, Z    +0.000, E1   +22.252, E3 +555744.779}
SPL {X  -162.820, Y  +608.428, Z    +0.000, E1   +22.255, E3 +555758.562}
SPL {X  -162.820, Y  +605.984, Z    +0.000, E1   +22.221, E3 +555771.199}
SPL {X  -162.820, Y  +603.020, Z    +0.000, E1   +22.272, E3 +555786.097}
SPL {X  -162.820, Y  +599.168, Z    +0.000, E1   +22.310, E3 +555805.365}
SPL {X  -162.820, Y  +596.569, Z    +0.000, E1   +22.222, E3 +555819.087}
SPL {X  -162.820, Y  +594.115, Z    +0.000, E1   +22.273, E3 +555831.313}
SPL {X  -162.820, Y  +591.721, Z    +0.000, E1   +22.239, E3 +555843.628}
SPL {X  -162.820, Y  +589.492, Z    +0.000, E1   +22.304, E3 +555854.489}
SPL {X  -162.820, Y  +587.447, Z    +0.000, E1   +22.279, E3 +555865.018}
SPL {X  -162.820, Y  +585.192, Z    +0.000, E1   +22.298, E3 +555876.428}
SPL {X  -162.820, Y  +582.610, Z    +0.000, E1   +22.234, E3 +555890.051}
SPL {X  -162.820, Y  +580.317, Z    +0.000, E1   +22.300, E3 +555901.105}
SPL {X  -162.820, Y  +578.878, Z    +0.000, E1   +22.272, E3 +555908.615}
SPL {X  -162.820, Y  +576.856, Z    +0.000, E1   +22.233, E3 +555919.373}
SPL {X  -162.820, Y  +573.830, Z    +0.000, E1   +22.272, E3 +555934.509}
SPL {X  -162.820, Y  +570.852, Z    +0.000, E1   +22.234, E3 +555949.968}
SPL {X  -162.820, Y  +568.608, Z    +0.000, E1   +22.253, E3 +555961.102}
SPL {X  -162.820, Y  +565.838, Z    +0.000, E1   +22.271, E3 +555975.333}
SPL {X  -162.820, Y  +562.162, Z    +0.000, E1   +22.252, E3 +555994.150}
SPL {X  -162.820, Y  +559.515, Z    +0.000, E1   +22.273, E3 +556007.269}
SPL {X  -162.820, Y  +556.723, Z    +0.000, E1   +22.309, E3 +556021.353}
SPL {X  -162.820, Y  +553.294, Z    +0.000, E1   +22.266, E3 +556039.140}
SPL {X  -162.820, Y  +550.871, Z    +0.000, E1   +22.229, E3 +556051.615}
SPL {X  -162.820, Y  +548.168, Z    +0.000, E1   +22.298, E3 +556064.951}
SPL {X  -162.820, Y  +545.860, Z    +0.000, E1   +22.216, E3 +556077.208}
SPL {X  -162.820, Y  +543.558, Z    +0.000, E1   +22.285, E3 +556088.439}
SPL {X  -162.820, Y  +540.968, Z    +0.000, E1   +22.274, E3 +556101.711}
SPL {X  -162.820, Y  +537.857, Z    +0.000, E1   +22.280, E3 +556117.587}
SPL {X  -162.820, Y  +534.880, Z    +0.000, E1   +22.252, E3 +556132.855}
SPL {X  -162.820, Y  +532.896, Z    +0.000, E1   +22.234, E3 +556143.016}
SPL {X  -162.820, Y  +531.056, Z    +0.000, E1   +22.251, E3 +556152.298}
SPL {X  -162.820, Y  +528.708, Z    +0.000, E1   +22.319, E3 +556163.679}
SPL {X  -162.820, Y  +526.907, Z    +0.000, E1   +22.243, E3 +556173.399}
SPL {X  -162.820, Y  +524.599, Z    +0.000, E1   +22.287, E3 +556184.922}
SPL {X  -162.820, Y  +522.011, Z    +0.000, E1   +22.282, E3 +556197.999}
SPL {X  -162.820, Y  +519.457, Z    +0.000, E1   +22.481, E3 +556209.288}
SPL {X  -162.820, Y  +505.859, Z    +0.000, E1   +28.367, E3 +556223.771}
SPL {X  -162.820, Y  +504.131, Z    +0.000, E1   +27.325, E3 +556237.910}
SPL {X  -162.820, Y  +503.215, Z    +0.000, E1   +26.369, E3 +556248.596}
SPL {X  -162.820, Y  +502.502, Z    +0.000, E1   +25.597, E3 +556257.442}
SPL {X  -162.820, Y  +501.672, Z    +0.000, E1   +24.583, E3 +556269.057}
SPL {X  -162.820, Y  +500.515, Z    +0.000, E1   +23.444, E3 +556283.587}
SPL {X  -162.820, Y  +499.633, Z    +0.000, E1   +22.486, E3 +556295.633}
SPL {X  -162.820, Y  +498.303, Z    +0.000, E1   +21.749, E3 +556308.943}
SPL {X  -162.820, Y  +495.897, Z    +0.000, E1   +21.662, E3 +556322.097}
SPL {X  -162.820, Y  +493.717, Z    +0.000, E1   +21.704, E3 +556333.203}
SPL {X  -162.820, Y  +491.396, Z    +0.000, E1   +21.707, E3 +556345.327}
SPL {X  -162.820, Y  +489.485, Z    +0.000, E1   +21.661, E3 +556355.675}
SPL {X  -162.820, Y  +487.723, Z    +0.000, E1   +21.665, E3 +556364.878}
SPL {X  -162.820, Y  +485.661, Z    +0.000, E1   +21.712, E3 +556375.322}
SPL {X  -162.820, Y  +482.775, Z    +0.000, E1   +21.716, E3 +556390.574}
SPL {X  -162.820, Y  +479.894, Z    +0.000, E1   +21.695, E3 +556405.650}
SPL {X  -162.820, Y  +477.685, Z    +0.000, E1   +21.656, E3 +556417.588}
SPL {X  -162.820, Y  +475.419, Z    +0.000, E1   +21.711, E3 +556428.940}
SPL {X  -162.820, Y  +473.301, Z    +0.000, E1   +21.712, E3 +556440.038}
SPL {X  -162.820, Y  +470.965, Z    +0.000, E1   +21.700, E3 +556452.383}
SPL {X  -162.820, Y  +469.036, Z    +0.000, E1   +21.695, E3 +556462.426}
SPL {X  -162.820, Y  +467.138, Z    +0.000, E1   +21.678, E3 +556472.598}
SPL {X  -162.820, Y  +465.011, Z    +0.000, E1   +21.692, E3 +556483.581}
SPL {X  -162.820, Y  +462.669, Z    +0.000, E1   +21.752, E3 +556495.361}
SPL {X  -162.820, Y  +460.725, Z    +0.000, E1   +21.689, E3 +556505.974}
SPL {X  -162.820, Y  +458.666, Z    +0.000, E1   +21.695, E3 +556516.786}
SPL {X  -162.820, Y  +456.431, Z    +0.000, E1   +21.708, E3 +556528.314}
SPL {X  -162.820, Y  +454.628, Z    +0.000, E1   +21.674, E3 +556538.033}
SPL {X  -162.820, Y  +452.690, Z    +0.000, E1   +21.773, E3 +556547.307}
SPL {X  -162.820, Y  +450.610, Z    +0.000, E1   +21.698, E3 +556558.906}
SPL {X  -162.820, Y  +448.170, Z    +0.000, E1   +21.667, E3 +556571.926}
SPL {X  -162.820, Y  +446.246, Z    +0.000, E1   +21.696, E3 +556581.744}
SPL {X  -162.820, Y  +443.784, Z    +0.000, E1   +21.713, E3 +556594.530}
SPL {X  -162.820, Y  +441.754, Z    +0.000, E1   +21.708, E3 +556605.082}
SPL {X  -162.820, Y  +439.933, Z    +0.000, E1   +21.690, E3 +556614.846}
SPL {X  -162.820, Y  +437.628, Z    +0.000, E1   +21.678, E3 +556627.034}
SPL {X  -162.820, Y  +435.262, Z    +0.000, E1   +21.727, E3 +556638.970}
SPL {X  -162.820, Y  +433.510, Z    +0.000, E1   +21.692, E3 +556648.384}
SPL {X  -162.820, Y  +431.492, Z    +0.000, E1   +21.686, E3 +556659.079}
SPL {X  -162.820, Y  +429.074, Z    +0.000, E1   +21.710, E3 +556671.531}
SPL {X  -162.820, Y  +427.020, Z    +0.000, E1   +21.674, E3 +556682.533}
SPL {X  -162.820, Y  +425.215, Z    +0.000, E1   +21.693, E3 +556691.835}
SPL {X  -162.820, Y  +422.986, Z    +0.000, E1   +21.685, E3 +556703.646}
SPL {X  -162.820, Y  +420.528, Z    +0.000, E1   +21.706, E3 +556716.296}
SPL {X  -162.820, Y  +418.116, Z    +0.000, E1   +21.761, E3 +556728.444}
SPL {X  -162.820, Y  +416.127, Z    +0.000, E1   +21.715, E3 +556739.149}
SPL {X  -162.820, Y  +414.361, Z    +0.000, E1   +21.613, E3 +556749.336}
SPL {X  -162.820, Y  +411.450, Z    +0.000, E1   +21.710, E3 +556763.910}
SPL {X  -162.820, Y  +408.590, Z    +0.000, E1   +21.735, E3 +556778.535}
SPL {X  -162.820, Y  +406.238, Z    +0.000, E1   +21.697, E3 +556791.184}
SPL {X  -162.820, Y  +403.166, Z    +0.000, E1   +21.746, E3 +556806.990}
SPL {X  -162.820, Y  +400.348, Z    +0.000, E1   +21.713, E3 +556821.825}
SPL {X  -162.820, Y  +398.298, Z    +0.000, E1   +21.721, E3 +556832.440}
SPL {X  -162.820, Y  +396.371, Z    +0.000, E1   +21.713, E3 +556842.622}
SPL {X  -162.820, Y  +394.508, Z    +0.000, E1   +21.616, E3 +556853.178}
SPL {X  -162.820, Y  +391.777, Z    +0.000, E1   +21.714, E3 +556866.837}
SPL {X  -162.820, Y  +388.822, Z    +0.000, E1   +21.717, E3 +556882.157}
SPL {X  -162.820, Y  +386.818, Z    +0.000, E1   +21.679, E3 +556892.897}
SPL {X  -162.820, Y  +384.697, Z    +0.000, E1   +21.693, E3 +556903.967}
SPL {X  -162.820, Y  +382.288, Z    +0.000, E1   +21.742, E3 +556916.090}
SPL {X  -162.817, Y  +379.520, Z    +0.000, E1   +21.723, E3 +556930.928}
SPL {X  -162.776, Y  +376.710, Z    +0.000, E1   +21.698, E3 +556945.667}
SPL {X  -162.707, Y  +374.438, Z    +0.000, E1   +21.688, E3 +556957.671}
SPL {X  -162.607, Y  +372.171, Z    +0.000, E1   +21.692, E3 +556969.470}
SPL {X  -162.494, Y  +370.197, Z    +0.000, E1   +21.655, E3 +556980.097}
SPL {X  -162.349, Y  +368.131, Z    +0.000, E1   +21.624, E3 +556991.215}
SPL {X  -162.161, Y  +365.866, Z    +0.000, E1   +21.642, E3 +557002.900}
SPL {X  -161.651, Y  +361.024, Z    +0.000, E1   +22.970, E3 +557016.323}
SPL {X  -160.281, Y  +351.857, Z    +0.000, E1   +24.243, E3 +557051.662}
ENDSPLINE

SPLINE
SPL {X  -161.833, Y  +362.603, Z    +0.000, E1   +17.021, E3 +557066.358}
ENDSPLINE

SPLINE
SPL {X  -160.786, Y  +354.842, Z    +0.000, E1   +19.274, E3 +557098.514}
ENDSPLINE

SPLINE
SPL {X  -162.485, Y  +370.062, Z    +0.000, E1   +10.606, E3 +557104.892}
SPL {X  -162.818, Y  +379.636, Z    +0.000, E1    +5.115, E3 +557094.241}
SPL {X  -162.820, Y  +386.976, Z    +0.000, E1    +0.144, E3 +557093.340}
SPL {X  -162.820, Y  +390.236, Z    +0.000, E1    -2.204, E3 +557099.398}
SPL {X  -162.820, Y  +393.415, Z    +0.000, E1    -4.587, E3 +557100.683}
SPL {X  -162.820, Y  +399.630, Z    +0.000, E1    -9.426, E3 +557102.612}
SPL {X  -162.820, Y  +408.127, Z    +0.000, E1   -18.417, E3 +557088.901}
SPL {X  -162.820, Y  +420.083, Z    +0.000, E1   -24.325, E3 +557109.376}
SPL {X  -162.820, Y  +428.527, Z    +0.000, E1   -26.988, E3 +557126.668}
SPL {X  -162.820, Y  +431.191, Z    +0.000, E1   -23.548, E3 +557161.521}
SPL {X  -162.820, Y  +432.946, Z    +0.000, E1   -22.795, E3 +557175.925}
SPL {X  -162.820, Y  +434.888, Z    +0.000, E1   -22.823, E3 +557185.331}
SPL {X  -162.820, Y  +436.834, Z    +0.000, E1   -22.779, E3 +557195.291}
SPL {X  -162.820, Y  +438.868, Z    +0.000, E1   -22.837, E3 +557204.945}
SPL {X  -162.820, Y  +441.351, Z    +0.000, E1   -22.805, E3 +557217.520}
SPL {X  -162.820, Y  +443.809, Z    +0.000, E1   -22.804, E3 +557229.687}
SPL {X  -162.820, Y  +447.077, Z    +0.000, E1   -22.869, E3 +557245.497}
SPL {X  -162.820, Y  +449.911, Z    +0.000, E1   -22.774, E3 +557260.107}
SPL {X  -162.820, Y  +451.861, Z    +0.000, E1   -22.750, E3 +557269.954}
SPL {X  -162.820, Y  +454.167, Z    +0.000, E1   -22.842, E3 +557280.684}
SPL {X  -162.820, Y  +456.529, Z    +0.000, E1   -22.855, E3 +557292.212}
SPL {X  -162.820, Y  +458.725, Z    +0.000, E1   -22.793, E3 +557303.616}
SPL {X  -162.820, Y  +460.754, Z    +0.000, E1   -22.806, E3 +557313.489}
SPL {X  -162.820, Y  +462.409, Z    +0.000, E1   -22.783, E3 +557321.906}
SPL {X  -162.820, Y  +464.633, Z    +0.000, E1   -22.813, E3 +557332.736}
SPL {X  -162.820, Y  +467.913, Z    +0.000, E1   -22.879, E3 +557348.575}
SPL {X  -162.820, Y  +470.892, Z    +0.000, E1   -22.837, E3 +557363.464}
SPL {X  -162.820, Y  +472.726, Z    +0.000, E1   -22.777, E3 +557373.003}
SPL {X  -162.820, Y  +475.118, Z    +0.000, E1   -22.777, E3 +557384.974}
SPL {X  -162.820, Y  +477.389, Z    +0.000, E1   -22.803, E3 +557395.891}
SPL {X  -162.820, Y  +478.914, Z    +0.000, E1   -22.821, E3 +557403.282}
SPL {X  -162.820, Y  +481.034, Z    +0.000, E1   -22.831, E3 +557413.804}
SPL {X  -162.820, Y  +484.256, Z    +0.000, E1   -22.840, E3 +557429.823}
SPL {X  -162.820, Y  +487.952, Z    +0.000, E1   -22.824, E3 +557448.253}
SPL {X  -162.820, Y  +491.768, Z    +0.000, E1   -22.852, E3 +557466.934}
SPL {X  -162.820, Y  +495.526, Z    +0.000, E1   -22.833, E3 +557485.705}
SPL {X  -162.820, Y  +499.330, Z    +0.000, E1   -22.841, E3 +557504.487}
SPL {X  -162.820, Y  +502.361, Z    +0.000, E1   -22.801, E3 +557519.645}
SPL {X  -162.820, Y  +505.323, Z    +0.000, E1   -22.838, E3 +557534.117}
SPL {X  -162.820, Y  +508.611, Z    +0.000, E1   -22.838, E3 +557550.380}
SPL {X  -162.820, Y  +511.620, Z    +0.000, E1   -22.791, E3 +557565.624}
SPL {X  -162.820, Y  +513.873, Z    +0.000, E1   -22.800, E3 +557576.596}
SPL {X  -162.820, Y  +516.100, Z    +0.000, E1   -22.809, E3 +557587.672}
SPL {X  -162.820, Y  +518.662, Z    +0.000, E1   -22.847, E3 +557599.971}
SPL {X  -162.820, Y  +520.641, Z    +0.000, E1   -22.790, E3 +557610.212}
SPL {X  -162.820, Y  +522.740, Z    +0.000, E1   -22.811, E3 +557620.454}
SPL {X  -162.820, Y  +524.628, Z    +0.000, E1   -22.846, E3 +557629.449}
SPL {X  -162.820, Y  +526.661, Z    +0.000, E1   -22.801, E3 +557640.005}
SPL {X  -162.820, Y  +529.662, Z    +0.000, E1   -22.810, E3 +557654.855}
SPL {X  -162.820, Y  +532.614, Z    +0.000, E1   -22.828, E3 +557669.262}
SPL {X  -162.820, Y  +534.838, Z    +0.000, E1   -22.864, E3 +557679.891}
SPL {X  -162.820, Y  +536.882, Z    +0.000, E1   -22.782, E3 +557690.745}
SPL {X  -162.820, Y  +539.194, Z    +0.000, E1   -22.826, E3 +557701.794}
SPL {X  -162.820, Y  +541.555, Z    +0.000, E1   -22.817, E3 +557713.608}
SPL {X  -162.820, Y  +543.728, Z    +0.000, E1   -22.799, E3 +557724.466}
SPL {X  -162.820, Y  +545.925, Z    +0.000, E1   -22.803, E3 +557735.336}
SPL {X  -162.820, Y  +549.071, Z    +0.000, E1   -22.836, E3 +557750.863}
SPL {X  -162.820, Y  +553.089, Z    +0.000, E1   -22.838, E3 +557770.763}
SPL {X  -162.820, Y  +556.430, Z    +0.000, E1   -22.821, E3 +557787.264}
SPL {X  -162.820, Y  +559.675, Z    +0.000, E1   -22.837, E3 +557803.344}
SPL {X  -162.820, Y  +562.799, Z    +0.000, E1   -22.814, E3 +557818.851}
SPL {X  -162.820, Y  +565.170, Z    +0.000, E1   -22.801, E3 +557830.676}
SPL {X  -162.820, Y  +568.020, Z    +0.000, E1   -22.787, E3 +557845.062}
SPL {X  -162.820, Y  +570.992, Z    +0.000, E1   -22.834, E3 +557859.281}
SPL {X  -162.820, Y  +572.901, Z    +0.000, E1   -22.775, E3 +557869.150}
SPL {X  -162.820, Y  +575.638, Z    +0.000, E1   -22.855, E3 +557882.259}
SPL {X  -162.820, Y  +578.553, Z    +0.000, E1   -22.801, E3 +557896.972}
SPL {X  -162.820, Y  +581.064, Z    +0.000, E1   -22.823, E3 +557909.256}
SPL {X  -162.820, Y  +583.435, Z    +0.000, E1   -22.808, E3 +557921.078}
SPL {X  -162.820, Y  +585.410, Z    +0.000, E1   -22.764, E3 +557931.213}
SPL {X  -162.820, Y  +587.676, Z    +0.000, E1   -22.853, E3 +557941.728}
SPL {X  -162.820, Y  +589.682, Z    +0.000, E1   -22.776, E3 +557952.258}
SPL {X  -162.820, Y  +591.720, Z    +0.000, E1   -22.868, E3 +557961.569}
SPL {X  -162.820, Y  +593.650, Z    +0.000, E1   -22.810, E3 +557971.639}
SPL {X  -162.820, Y  +595.830, Z    +0.000, E1   -22.828, E3 +557982.254}
SPL {X  -162.820, Y  +598.094, Z    +0.000, E1   -22.843, E3 +557993.368}
SPL {X  -162.820, Y  +600.420, Z    +0.000, E1   -22.826, E3 +558004.999}
SPL {X  -162.820, Y  +602.573, Z    +0.000, E1   -22.830, E3 +558015.584}
SPL {X  -162.820, Y  +604.828, Z    +0.000, E1   -22.784, E3 +558027.222}
SPL {X  -162.820, Y  +608.133, Z    +0.000, E1   -22.831, E3 +558043.340}
SPL {X  -162.820, Y  +611.103, Z    +0.000, E1   -22.785, E3 +558058.266}
SPL {X  -162.820, Y  +613.294, Z    +0.000, E1   -22.780, E3 +558069.139}
SPL {X  -162.820, Y  +615.356, Z    +0.000, E1   -22.799, E3 +558079.196}
SPL {X  -162.820, Y  +617.439, Z    +0.000, E1   -22.808, E3 +558089.454}
SPL {X  -162.820, Y  +619.665, Z    +0.000, E1   -22.817, E3 +558100.422}
SPL {X  -162.820, Y  +621.733, Z    +0.000, E1   -22.759, E3 +558111.146}
SPL {X  -162.820, Y  +624.076, Z    +0.000, E1   -22.774, E3 +558122.652}
SPL {X  -162.820, Y  +627.244, Z    +0.000, E1   -22.803, E3 +558138.334}
SPL {X  -162.820, Y  +630.349, Z    +0.000, E1   -22.766, E3 +558153.866}
SPL {X  -162.820, Y  +632.572, Z    +0.000, E1   -22.785, E3 +558164.672}
SPL {X  -162.820, Y  +634.507, Z    +0.000, E1   -22.784, E3 +558174.311}
SPL {X  -162.820, Y  +636.863, Z    +0.000, E1   -22.760, E3 +558186.233}
SPL {X  -162.820, Y  +640.111, Z    +0.000, E1   -22.809, E3 +558202.116}
SPL {X  -162.820, Y  +643.449, Z    +0.000, E1   -22.796, E3 +558218.634}
SPL {X  -162.820, Y  +645.630, Z    +0.000, E1   -22.795, E3 +558229.330}
SPL {X  -162.820, Y  +647.561, Z    +0.000, E1   -22.705, E3 +558239.781}
SPL {X  -162.820, Y  +651.051, Z    +0.000, E1   -22.833, E3 +558256.200}
SPL {X  -162.820, Y  +653.898, Z    +0.000, E1   -22.796, E3 +558270.386}
SPL {X  -162.820, Y  +656.161, Z    +0.000, E1   -22.812, E3 +558281.507}
SPL {X  -162.820, Y  +658.384, Z    +0.000, E1   -22.822, E3 +558292.374}
SPL {X  -162.820, Y  +660.215, Z    +0.000, E1   -22.649, E3 +558302.964}
SPL {X  -162.820, Y  +662.823, Z    +0.000, E1   -22.799, E3 +558314.672}
SPL {X  -162.820, Y  +665.112, Z    +0.000, E1   -22.835, E3 +558325.727}
SPL {X  -162.820, Y  +667.016, Z    +0.000, E1   -22.823, E3 +558335.155}
SPL {X  -162.820, Y  +668.960, Z    +0.000, E1   -22.773, E3 +558345.323}
SPL {X  -162.820, Y  +672.333, Z    +0.000, E1   -22.837, E3 +558361.659}
SPL {X  -162.812, Y  +675.071, Z    +0.000, E1   -22.742, E3 +558375.804}
SPL {X  -162.773, Y  +677.428, Z    +0.000, E1   -22.762, E3 +558387.401}
SPL {X  -162.691, Y  +679.987, Z    +0.000, E1   -22.794, E3 +558399.815}
SPL {X  -162.559, Y  +682.717, Z    +0.000, E1   -22.726, E3 +558413.998}
SPL {X  -162.404, Y  +685.137, Z    +0.000, E1   -22.766, E3 +558425.520}
SPL {X  -162.229, Y  +687.364, Z    +0.000, E1   -22.685, E3 +558437.389}
SPL {X  -161.938, Y  +690.422, Z    +0.000, E1   -22.769, E3 +558451.795}
SPL {X  -161.065, Y  +697.344, Z    +0.000, E1   -25.698, E3 +558460.914}
SPL {X  -158.730, Y  +709.763, Z    +0.000, E1   -31.225, E3 +558469.588}
ENDSPLINE

SPLINE
SPL {X  -160.932, Y  +698.225, Z    +0.000, E1   -21.712, E3 +558500.697}
SPL {X  -161.691, Y  +692.643, Z    +0.000, E1   -17.369, E3 +558517.580}
SPL {X  -162.534, Y  +683.153, Z    +0.000, E1   -10.475, E3 +558543.047}
SPL {X  -162.820, Y  +670.105, Z    +0.000, E1    -2.484, E3 +558535.694}
SPL {X  -162.820, Y  +665.819, Z    +0.000, E1    +0.492, E3 +558537.990}
SPL {X  -162.820, Y  +661.883, Z    +0.000, E1    +3.373, E3 +558542.466}
SPL {X  -162.820, Y  +655.163, Z    +0.000, E1    +8.702, E3 +558542.065}
SPL {X  -162.820, Y  +634.515, Z    +0.000, E1   +26.439, E3 +558534.478}
ENDSPLINE

SPLINE
SPL {X  -162.820, Y  +638.080, Z    +0.000, E1   +18.858, E3 +558564.443}
ENDSPLINE

SPLINE
SPL {X  -162.820, Y  +623.278, Z    +0.000, E1   +28.723, E3 +558566.013}
SPL {X  -162.820, Y  +618.658, Z    +0.000, E1   +26.841, E3 +558594.622}
ENDSPLINE

SPLINE
SPL {X  -162.820, Y  +623.685, Z    +0.000, E1   +22.346, E3 +558606.929}
ENDSPLINE

SPLINE
SPL {X  -162.820, Y  +621.304, Z    +0.000, E1   +22.259, E3 +558619.744}
SPL {X  -162.820, Y  +618.758, Z    +0.000, E1   +22.239, E3 +558632.895}
SPL {X  -162.820, Y  +616.062, Z    +0.000, E1   +22.275, E3 +558646.316}
SPL {X  -162.820, Y  +613.536, Z    +0.000, E1   +22.242, E3 +558659.437}
SPL {X  -162.820, Y  +611.128, Z    +0.000, E1   +22.252, E3 +558671.608}
SPL {X  -162.820, Y  +608.428, Z    +0.000, E1   +22.255, E3 +558685.391}
SPL {X  -162.820, Y  +605.984, Z    +0.000, E1   +22.221, E3 +558698.028}
SPL {X  -162.820, Y  +603.020, Z    +0.000, E1   +22.272, E3 +558712.927}
SPL {X  -162.820, Y  +599.842, Z    +0.000, E1   +22.298, E3 +558728.692}
SPL {X  -162.820, Y  +597.194, Z    +0.000, E1   +22.253, E3 +558742.613}
SPL {X  -162.820, Y  +594.779, Z    +0.000, E1   +22.284, E3 +558754.517}
SPL {X  -162.820, Y  +592.389, Z    +0.000, E1   +22.245, E3 +558767.134}
SPL {X  -162.820, Y  +589.492, Z    +0.000, E1   +22.304, E3 +558781.318}
SPL {X  -162.820, Y  +587.447, Z    +0.000, E1   +22.279, E3 +558791.847}
SPL {X  -162.820, Y  +585.192, Z    +0.000, E1   +22.298, E3 +558803.257}
SPL {X  -162.820, Y  +582.610, Z    +0.000, E1   +22.234, E3 +558816.881}
SPL {X  -162.820, Y  +579.691, Z    +0.000, E1   +22.312, E3 +558831.152}
SPL {X  -162.820, Y  +577.460, Z    +0.000, E1   +22.218, E3 +558843.139}
SPL {X  -162.820, Y  +575.394, Z    +0.000, E1   +22.240, E3 +558853.564}
SPL {X  -162.820, Y  +572.645, Z    +0.000, E1   +22.246, E3 +558867.561}
SPL {X  -162.820, Y  +570.282, Z    +0.000, E1   +22.231, E3 +558879.612}
SPL {X  -162.820, Y  +567.961, Z    +0.000, E1   +22.247, E3 +558891.401}
SPL {X  -162.820, Y  +564.506, Z    +0.000, E1   +22.298, E3 +558908.716}
SPL {X  -162.820, Y  +561.620, Z    +0.000, E1   +22.191, E3 +558924.097}
SPL {X  -162.820, Y  +559.515, Z    +0.000, E1   +22.273, E3 +558934.098}
SPL {X  -162.820, Y  +556.723, Z    +0.000, E1   +22.309, E3 +558948.182}
SPL {X  -162.820, Y  +554.378, Z    +0.000, E1   +22.288, E3 +558960.027}
SPL {X  -162.820, Y  +552.787, Z    +0.000, E1   +22.213, E3 +558968.849}
SPL {X  -162.820, Y  +550.871, Z    +0.000, E1   +22.229, E3 +558978.444}
SPL {X  -162.820, Y  +548.168, Z    +0.000, E1   +22.298, E3 +558991.780}
SPL {X  -162.820, Y  +545.860, Z    +0.000, E1   +22.216, E3 +559004.038}
SPL {X  -162.820, Y  +543.558, Z    +0.000, E1   +22.285, E3 +559015.268}
SPL {X  -162.820, Y  +540.968, Z    +0.000, E1   +22.274, E3 +559028.541}
SPL {X  -162.820, Y  +538.512, Z    +0.000, E1   +22.287, E3 +559040.853}
SPL {X  -162.820, Y  +535.523, Z    +0.000, E1   +22.266, E3 +559056.468}
SPL {X  -162.820, Y  +531.757, Z    +0.000, E1   +22.276, E3 +559075.523}
SPL {X  -162.820, Y  +527.980, Z    +0.000, E1   +22.326, E3 +559094.354}
SPL {X  -162.820, Y  +524.599, Z    +0.000, E1   +22.287, E3 +559111.751}
SPL {X  -162.820, Y  +522.011, Z    +0.000, E1   +22.282, E3 +559124.828}
SPL {X  -162.820, Y  +519.457, Z    +0.000, E1   +22.481, E3 +559136.118}
SPL {X  -162.820, Y  +505.859, Z    +0.000, E1   +28.367, E3 +559150.601}
SPL {X  -162.820, Y  +504.131, Z    +0.000, E1   +27.325, E3 +559164.739}
SPL {X  -162.820, Y  +502.813, Z    +0.000, E1   +26.013, E3 +559180.115}
SPL {X  -162.820, Y  +502.016, Z    +0.000, E1   +24.802, E3 +559192.458}
SPL {X  -162.820, Y  +501.060, Z    +0.000, E1   +24.081, E3 +559202.647}
SPL {X  -162.820, Y  +499.934, Z    +0.000, E1   +22.814, E3 +559218.516}
SPL {X  -162.820, Y  +498.303, Z    +0.000, E1   +21.749, E3 +559235.772}
SPL {X  -162.820, Y  +495.897, Z    +0.000, E1   +21.662, E3 +559248.926}
SPL {X  -162.820, Y  +493.717, Z    +0.000, E1   +21.704, E3 +559260.032}
SPL {X  -162.820, Y  +491.396, Z    +0.000, E1   +21.707, E3 +559272.156}
SPL {X  -162.820, Y  +489.485, Z    +0.000, E1   +21.661, E3 +559282.504}
SPL {X  -162.820, Y  +487.723, Z    +0.000, E1   +21.665, E3 +559291.707}
SPL {X  -162.820, Y  +485.661, Z    +0.000, E1   +21.712, E3 +559302.151}
SPL {X  -162.820, Y  +482.775, Z    +0.000, E1   +21.716, E3 +559317.403}
SPL {X  -162.820, Y  +479.894, Z    +0.000, E1   +21.695, E3 +559332.480}
SPL {X  -162.820, Y  +477.685, Z    +0.000, E1   +21.656, E3 +559344.417}
SPL {X  -162.820, Y  +475.419, Z    +0.000, E1   +21.711, E3 +559355.770}
SPL {X  -162.820, Y  +473.301, Z    +0.000, E1   +21.712, E3 +559366.867}
SPL {X  -162.820, Y  +470.965, Z    +0.000, E1   +21.700, E3 +559379.212}
SPL {X  -162.820, Y  +469.036, Z    +0.000, E1   +21.695, E3 +559389.256}
SPL {X  -162.820, Y  +467.138, Z    +0.000, E1   +21.678, E3 +559399.427}
SPL {X  -162.820, Y  +465.011, Z    +0.000, E1   +21.692, E3 +559410.410}
SPL {X  -162.820, Y  +462.669, Z    +0.000, E1   +21.752, E3 +559422.190}
SPL {X  -162.820, Y  +460.725, Z    +0.000, E1   +21.689, E3 +559432.803}
SPL {X  -162.820, Y  +458.666, Z    +0.000, E1   +21.695, E3 +559443.615}
SPL {X  -162.820, Y  +456.431, Z    +0.000, E1   +21.708, E3 +559455.144}
SPL {X  -162.820, Y  +453.609, Z    +0.000, E1   +21.757, E3 +559469.678}
SPL {X  -162.820, Y  +450.610, Z    +0.000, E1   +21.698, E3 +559485.735}
SPL {X  -162.820, Y  +448.170, Z    +0.000, E1   +21.667, E3 +559498.756}
SPL {X  -162.820, Y  +446.246, Z    +0.000, E1   +21.696, E3 +559508.573}
SPL {X  -162.820, Y  +443.784, Z    +0.000, E1   +21.713, E3 +559521.360}
SPL {X  -162.820, Y  +440.567, Z    +0.000, E1   +21.731, E3 +559538.199}
SPL {X  -162.820, Y  +437.628, Z    +0.000, E1   +21.678, E3 +559553.864}
SPL {X  -162.820, Y  +435.262, Z    +0.000, E1   +21.727, E3 +559565.799}
SPL {X  -162.820, Y  +433.510, Z    +0.000, E1   +21.692, E3 +559575.213}
SPL {X  -162.820, Y  +431.492, Z    +0.000, E1   +21.686, E3 +559585.908}
SPL {X  -162.820, Y  +429.074, Z    +0.000, E1   +21.710, E3 +559598.360}
SPL {X  -162.820, Y  +427.020, Z    +0.000, E1   +21.674, E3 +559609.362}
SPL {X  -162.820, Y  +424.525, Z    +0.000, E1   +21.712, E3 +559622.275}
SPL {X  -162.820, Y  +421.144, Z    +0.000, E1   +21.719, E3 +559639.942}
SPL {X  -162.820, Y  +418.116, Z    +0.000, E1   +21.761, E3 +559655.273}
SPL {X  -162.820, Y  +416.127, Z    +0.000, E1   +21.715, E3 +559665.978}
SPL {X  -162.820, Y  +414.361, Z    +0.000, E1   +21.613, E3 +559676.165}
SPL {X  -162.820, Y  +412.134, Z    +0.000, E1   +21.697, E3 +559687.110}
SPL {X  -162.820, Y  +409.248, Z    +0.000, E1   +21.741, E3 +559702.045}
SPL {X  -162.820, Y  +406.238, Z    +0.000, E1   +21.697, E3 +559718.013}
SPL {X  -162.820, Y  +404.001, Z    +0.000, E1   +21.723, E3 +559729.443}
SPL {X  -162.820, Y  +402.223, Z    +0.000, E1   +21.697, E3 +559738.928}
SPL {X  -162.820, Y  +400.348, Z    +0.000, E1   +21.713, E3 +559748.654}
SPL {X  -162.820, Y  +398.298, Z    +0.000, E1   +21.721, E3 +559759.270}
SPL {X  -162.820, Y  +396.371, Z    +0.000, E1   +21.713, E3 +559769.451}
SPL {X  -162.820, Y  +394.508, Z    +0.000, E1   +21.616, E3 +559780.007}
SPL {X  -162.820, Y  +392.435, Z    +0.000, E1   +21.681, E3 +559790.360}
SPL {X  -162.820, Y  +389.390, Z    +0.000, E1   +21.742, E3 +559805.967}
SPL {X  -162.820, Y  +386.818, Z    +0.000, E1   +21.679, E3 +559819.726}
SPL {X  -162.820, Y  +384.697, Z    +0.000, E1   +21.693, E3 +559830.796}
SPL {X  -162.820, Y  +382.288, Z    +0.000, E1   +21.742, E3 +559842.920}
SPL {X  -162.820, Y  +380.381, Z    +0.000, E1   +21.655, E3 +559853.645}
SPL {X  -162.808, Y  +378.512, Z    +0.000, E1   +21.736, E3 +559862.697}
SPL {X  -162.776, Y  +376.710, Z    +0.000, E1   +21.698, E3 +559872.496}
SPL {X  -162.707, Y  +374.438, Z    +0.000, E1   +21.688, E3 +559884.500}
SPL {X  -162.607, Y  +372.171, Z    +0.000, E1   +21.692, E3 +559896.300}
SPL {X  -162.494, Y  +370.197, Z    +0.000, E1   +21.655, E3 +559906.926}
SPL {X  -162.349, Y  +368.131, Z    +0.000, E1   +21.624, E3 +559918.044}
SPL {X  -162.161, Y  +365.866, Z    +0.000, E1   +21.642, E3 +559929.729}
SPL {X  -161.927, Y  +363.466, Z    +0.000, E1   +21.730, E3 +559941.501}
SPL {X  -160.290, Y  +351.907, Z    +0.000, E1   +27.562, E3 +559949.078}
SPL {X  -159.725, Y  +348.905, Z    +0.000, E1   +26.136, E3 +559974.314}
ENDSPLINE

SPLINE
SPL {X  -160.871, Y  +355.385, Z    +0.000, E1   +21.841, E3 +559983.157}
SPL {X  -161.833, Y  +362.603, Z    +0.000, E1   +17.021, E3 +559993.187}
ENDSPLINE

SPLINE
SPL {X  -160.786, Y  +354.842, Z    +0.000, E1   +19.274, E3 +560025.343}
ENDSPLINE

SPLINE
SPL {X  -162.485, Y  +370.062, Z    +0.000, E1   +10.606, E3 +560031.721}
SPL {X  -162.818, Y  +379.636, Z    +0.000, E1    +5.115, E3 +560021.070}
SPL {X  -162.820, Y  +386.976, Z    +0.000, E1    +0.144, E3 +560020.169}
SPL {X  -162.820, Y  +391.982, Z    +0.000, E1    -3.443, E3 +560026.934}
SPL {X  -162.820, Y  +399.630, Z    +0.000, E1    -9.426, E3 +560029.441}
SPL {X  -162.820, Y  +408.127, Z    +0.000, E1   -18.417, E3 +560015.730}
SPL {X  -162.820, Y  +420.083, Z    +0.000, E1   -24.325, E3 +560036.205}
SPL {X  -162.820, Y  +428.527, Z    +0.000, E1   -26.988, E3 +560053.497}
SPL {X  -162.820, Y  +431.336, Z    +0.000, E1   -24.162, E3 +560083.707}
SPL {X  -162.820, Y  +432.048, Z    +0.000, E1   -22.832, E3 +560098.211}
SPL {X  -162.820, Y  +434.888, Z    +0.000, E1   -22.823, E3 +560112.161}
SPL {X  -162.820, Y  +436.834, Z    +0.000, E1   -22.779, E3 +560122.121}
SPL {X  -162.820, Y  +438.868, Z    +0.000, E1   -22.837, E3 +560131.774}
SPL {X  -162.820, Y  +441.351, Z    +0.000, E1   -22.805, E3 +560144.350}
SPL {X  -162.820, Y  +443.809, Z    +0.000, E1   -22.804, E3 +560156.516}
SPL {X  -162.820, Y  +446.105, Z    +0.000, E1   -22.815, E3 +560167.758}
SPL {X  -162.820, Y  +447.974, Z    +0.000, E1   -22.856, E3 +560176.661}
SPL {X  -162.820, Y  +449.911, Z    +0.000, E1   -22.774, E3 +560186.936}
SPL {X  -162.820, Y  +451.861, Z    +0.000, E1   -22.750, E3 +560196.783}
SPL {X  -162.820, Y  +454.167, Z    +0.000, E1   -22.842, E3 +560207.513}
SPL {X  -162.820, Y  +456.529, Z    +0.000, E1   -22.855, E3 +560219.041}
SPL {X  -162.820, Y  +458.725, Z    +0.000, E1   -22.793, E3 +560230.446}
SPL {X  -162.820, Y  +461.700, Z    +0.000, E1   -22.822, E3 +560245.068}
SPL {X  -162.820, Y  +464.633, Z    +0.000, E1   -22.813, E3 +560259.565}
SPL {X  -162.820, Y  +466.699, Z    +0.000, E1   -22.824, E3 +560269.611}
SPL {X  -162.820, Y  +468.655, Z    +0.000, E1   -22.858, E3 +560279.055}
SPL {X  -162.820, Y  +470.892, Z    +0.000, E1   -22.837, E3 +560290.293}
SPL {X  -162.820, Y  +472.726, Z    +0.000, E1   -22.777, E3 +560299.832}
SPL {X  -162.820, Y  +475.118, Z    +0.000, E1   -22.777, E3 +560311.803}
SPL {X  -162.820, Y  +478.177, Z    +0.000, E1   -22.834, E3 +560326.496}
SPL {X  -162.820, Y  +481.034, Z    +0.000, E1   -22.831, E3 +560340.634}
SPL {X  -162.820, Y  +483.391, Z    +0.000, E1   -22.793, E3 +560352.570}
SPL {X  -162.820, Y  +486.307, Z    +0.000, E1   -22.833, E3 +560366.824}
SPL {X  -162.820, Y  +488.828, Z    +0.000, E1   -22.793, E3 +560379.466}
SPL {X  -162.820, Y  +491.768, Z    +0.000, E1   -22.852, E3 +560393.764}
SPL {X  -162.820, Y  +495.526, Z    +0.000, E1   -22.833, E3 +560412.535}
SPL {X  -162.820, Y  +499.330, Z    +0.000, E1   -22.841, E3 +560431.316}
SPL {X  -162.820, Y  +503.049, Z    +0.000, E1   -22.823, E3 +560449.865}
SPL {X  -162.820, Y  +505.970, Z    +0.000, E1   -22.835, E3 +560464.038}
SPL {X  -162.820, Y  +508.611, Z    +0.000, E1   -22.838, E3 +560477.209}
SPL {X  -162.820, Y  +511.620, Z    +0.000, E1   -22.791, E3 +560492.453}
SPL {X  -162.820, Y  +513.873, Z    +0.000, E1   -22.800, E3 +560503.425}
SPL {X  -162.820, Y  +516.100, Z    +0.000, E1   -22.809, E3 +560514.501}
SPL {X  -162.820, Y  +518.662, Z    +0.000, E1   -22.847, E3 +560526.800}
SPL {X  -162.820, Y  +520.641, Z    +0.000, E1   -22.790, E3 +560537.041}
SPL {X  -162.820, Y  +522.740, Z    +0.000, E1   -22.811, E3 +560547.284}
SPL {X  -162.820, Y  +525.255, Z    +0.000, E1   -22.822, E3 +560559.704}
SPL {X  -162.820, Y  +528.050, Z    +0.000, E1   -22.808, E3 +560573.669}
SPL {X  -162.820, Y  +530.303, Z    +0.000, E1   -22.798, E3 +560584.823}
SPL {X  -162.820, Y  +532.614, Z    +0.000, E1   -22.828, E3 +560596.091}
SPL {X  -162.820, Y  +534.838, Z    +0.000, E1   -22.864, E3 +560606.720}
SPL {X  -162.820, Y  +536.882, Z    +0.000, E1   -22.782, E3 +560617.575}
SPL {X  -162.820, Y  +539.194, Z    +0.000, E1   -22.826, E3 +560628.623}
SPL {X  -162.820, Y  +541.555, Z    +0.000, E1   -22.817, E3 +560640.438}
SPL {X  -162.820, Y  +543.728, Z    +0.000, E1   -22.799, E3 +560651.295}
SPL {X  -162.820, Y  +545.925, Z    +0.000, E1   -22.803, E3 +560662.165}
SPL {X  -162.820, Y  +549.071, Z    +0.000, E1   -22.836, E3 +560677.692}
SPL {X  -162.820, Y  +553.089, Z    +0.000, E1   -22.838, E3 +560697.592}
SPL {X  -162.820, Y  +556.430, Z    +0.000, E1   -22.821, E3 +560714.093}
SPL {X  -162.820, Y  +558.974, Z    +0.000, E1   -22.806, E3 +560726.793}
SPL {X  -162.820, Y  +562.171, Z    +0.000, E1   -22.845, E3 +560742.492}
SPL {X  -162.820, Y  +565.170, Z    +0.000, E1   -22.801, E3 +560757.505}
SPL {X  -162.820, Y  +567.308, Z    +0.000, E1   -22.750, E3 +560768.521}
SPL {X  -162.820, Y  +570.378, Z    +0.000, E1   -22.843, E3 +560783.145}
SPL {X  -162.820, Y  +573.634, Z    +0.000, E1   -22.827, E3 +560799.289}
SPL {X  -162.820, Y  +576.228, Z    +0.000, E1   -22.814, E3 +560812.185}
SPL {X  -162.820, Y  +578.553, Z    +0.000, E1   -22.801, E3 +560823.801}
SPL {X  -162.820, Y  +581.064, Z    +0.000, E1   -22.823, E3 +560836.085}
SPL {X  -162.820, Y  +583.435, Z    +0.000, E1   -22.808, E3 +560847.907}
SPL {X  -162.820, Y  +585.410, Z    +0.000, E1   -22.764, E3 +560858.043}
SPL {X  -162.820, Y  +587.676, Z    +0.000, E1   -22.853, E3 +560868.557}
SPL {X  -162.820, Y  +589.682, Z    +0.000, E1   -22.776, E3 +560879.087}
SPL {X  -162.820, Y  +591.720, Z    +0.000, E1   -22.868, E3 +560888.398}
SPL {X  -162.820, Y  +593.650, Z    +0.000, E1   -22.810, E3 +560898.468}
SPL {X  -162.820, Y  +595.830, Z    +0.000, E1   -22.828, E3 +560909.084}
SPL {X  -162.820, Y  +598.094, Z    +0.000, E1   -22.843, E3 +560920.197}
SPL {X  -162.820, Y  +600.420, Z    +0.000, E1   -22.826, E3 +560931.828}
SPL {X  -162.820, Y  +602.573, Z    +0.000, E1   -22.830, E3 +560942.413}
SPL {X  -162.820, Y  +604.828, Z    +0.000, E1   -22.784, E3 +560954.052}
SPL {X  -162.820, Y  +607.142, Z    +0.000, E1   -22.808, E3 +560965.232}
SPL {X  -162.820, Y  +608.890, Z    +0.000, E1   -22.790, E3 +560974.057}
SPL {X  -162.820, Y  +611.103, Z    +0.000, E1   -22.785, E3 +560985.095}
SPL {X  -162.820, Y  +613.294, Z    +0.000, E1   -22.780, E3 +560995.968}
SPL {X  -162.820, Y  +615.356, Z    +0.000, E1   -22.799, E3 +561006.025}
SPL {X  -162.820, Y  +617.439, Z    +0.000, E1   -22.808, E3 +561016.284}
SPL {X  -162.820, Y  +619.665, Z    +0.000, E1   -22.817, E3 +561027.252}
SPL {X  -162.820, Y  +621.733, Z    +0.000, E1   -22.759, E3 +561037.976}
SPL {X  -162.820, Y  +624.076, Z    +0.000, E1   -22.774, E3 +561049.481}
SPL {X  -162.820, Y  +626.527, Z    +0.000, E1   -22.768, E3 +561061.723}
SPL {X  -162.820, Y  +629.758, Z    +0.000, E1   -22.800, E3 +561077.652}
SPL {X  -162.820, Y  +632.572, Z    +0.000, E1   -22.785, E3 +561091.502}
SPL {X  -162.820, Y  +634.507, Z    +0.000, E1   -22.784, E3 +561101.140}
SPL {X  -162.820, Y  +636.863, Z    +0.000, E1   -22.760, E3 +561113.063}
SPL {X  -162.820, Y  +639.254, Z    +0.000, E1   -22.767, E3 +561124.846}
SPL {X  -162.820, Y  +641.195, Z    +0.000, E1   -22.782, E3 +561134.294}
SPL {X  -162.820, Y  +643.449, Z    +0.000, E1   -22.796, E3 +561145.463}
SPL {X  -162.820, Y  +645.630, Z    +0.000, E1   -22.795, E3 +561156.159}
SPL {X  -162.820, Y  +647.561, Z    +0.000, E1   -22.705, E3 +561166.610}
SPL {X  -162.820, Y  +651.051, Z    +0.000, E1   -22.833, E3 +561183.029}
SPL {X  -162.820, Y  +653.898, Z    +0.000, E1   -22.796, E3 +561197.215}
SPL {X  -162.820, Y  +656.161, Z    +0.000, E1   -22.812, E3 +561208.337}
SPL {X  -162.820, Y  +658.384, Z    +0.000, E1   -22.822, E3 +561219.203}
SPL {X  -162.820, Y  +660.215, Z    +0.000, E1   -22.649, E3 +561229.794}
SPL {X  -162.820, Y  +662.823, Z    +0.000, E1   -22.799, E3 +561241.502}
SPL {X  -162.820, Y  +665.112, Z    +0.000, E1   -22.835, E3 +561252.556}
SPL {X  -162.820, Y  +667.016, Z    +0.000, E1   -22.823, E3 +561261.984}
SPL {X  -162.820, Y  +668.960, Z    +0.000, E1   -22.773, E3 +561272.152}
SPL {X  -162.820, Y  +672.333, Z    +0.000, E1   -22.837, E3 +561288.488}
SPL {X  -162.812, Y  +675.071, Z    +0.000, E1   -22.742, E3 +561302.633}
SPL {X  -162.773, Y  +677.428, Z    +0.000, E1   -22.762, E3 +561314.230}
SPL {X  -162.691, Y  +679.987, Z    +0.000, E1   -22.794, E3 +561326.644}
SPL {X  -162.604, Y  +681.880, Z    +0.000, E1   -22.691, E3 +561336.804}
SPL {X  -162.458, Y  +684.346, Z    +0.000, E1   -22.764, E3 +561348.598}
SPL {X  -162.296, Y  +686.547, Z    +0.000, E1   -22.660, E3 +561360.215}
SPL {X  -162.090, Y  +688.902, Z    +0.000, E1   -22.700, E3 +561371.723}
SPL {X  -161.474, Y  +694.390, Z    +0.000, E1   -24.298, E3 +561385.078}
SPL {X  -158.730, Y  +709.763, Z    +0.000, E1   -31.225, E3 +561396.417}
ENDSPLINE

SPLINE
SPL {X  -160.932, Y  +698.225, Z    +0.000, E1   -21.712, E3 +561427.526}
SPL {X  -161.917, Y  +690.622, Z    +0.000, E1   -16.445, E3 +561441.127}
ENDSPLINE

SPLINE
SPL {X  -161.349, Y  +695.340, Z    +0.000, E1   -18.625, E3 +561448.745}
ENDSPLINE

SPLINE
SPL {X  -162.534, Y  +683.153, Z    +0.000, E1   -10.475, E3 +561469.876}
SPL {X  -162.820, Y  +667.630, Z    +0.000, E1    -0.882, E3 +561463.853}
SPL {X  -162.820, Y  +661.883, Z    +0.000, E1    +3.373, E3 +561469.296}
SPL {X  -162.820, Y  +653.808, Z    +0.000, E1    +9.891, E3 +561466.987}
SPL {X  -162.820, Y  +632.548, Z    +0.000, E1   +27.446, E3 +561463.524}
ENDSPLINE

SPLINE
SPL {X  -162.820, Y  +638.080, Z    +0.000, E1   +18.858, E3 +561491.272}
ENDSPLINE

SPLINE
SPL {X  -162.820, Y  +623.278, Z    +0.000, E1   +28.723, E3 +561492.843}
SPL {X  -162.820, Y  +618.658, Z    +0.000, E1   +26.841, E3 +561521.452}
ENDSPLINE

SPLINE
SPL {X  -162.820, Y  +623.685, Z    +0.000, E1   +22.346, E3 +561533.758}
ENDSPLINE

SPLINE
SPL {X  -162.820, Y  +621.304, Z    +0.000, E1   +22.259, E3 +561546.574}
SPL {X  -162.820, Y  +618.758, Z    +0.000, E1   +22.239, E3 +561559.724}
SPL {X  -162.820, Y  +616.062, Z    +0.000, E1   +22.275, E3 +561573.145}
SPL {X  -162.820, Y  +613.536, Z    +0.000, E1   +22.242, E3 +561586.266}
SPL {X  -162.820, Y  +610.461, Z    +0.000, E1   +22.264, E3 +561601.898}
SPL {X  -162.820, Y  +606.755, Z    +0.000, E1   +22.275, E3 +561620.696}
SPL {X  -162.820, Y  +603.020, Z    +0.000, E1   +22.272, E3 +561639.756}
SPL {X  -162.820, Y  +599.168, Z    +0.000, E1   +22.310, E3 +561659.024}
SPL {X  -162.820, Y  +595.597, Z    +0.000, E1   +22.284, E3 +561677.360}
SPL {X  -162.820, Y  +593.320, Z    +0.000, E1   +22.199, E3 +561689.450}
SPL {X  -162.820, Y  +591.031, Z    +0.000, E1   +22.283, E3 +561700.541}
SPL {X  -162.820, Y  +588.026, Z    +0.000, E1   +22.301, E3 +561715.668}
SPL {X  -162.820, Y  +585.899, Z    +0.000, E1   +22.286, E3 +561726.470}
SPL {X  -162.820, Y  +583.204, Z    +0.000, E1   +22.278, E3 +561740.493}
SPL {X  -162.820, Y  +579.691, Z    +0.000, E1   +22.312, E3 +561757.981}
SPL {X  -162.820, Y  +576.856, Z    +0.000, E1   +22.233, E3 +561773.032}
SPL {X  -162.820, Y  +574.811, Z    +0.000, E1   +22.236, E3 +561783.295}
SPL {X  -162.820, Y  +572.645, Z    +0.000, E1   +22.246, E3 +561794.391}
SPL {X  -162.820, Y  +569.475, Z    +0.000, E1   +22.269, E3 +561810.397}
SPL {X  -162.820, Y  +565.838, Z    +0.000, E1   +22.271, E3 +561828.992}
SPL {X  -162.820, Y  +562.162, Z    +0.000, E1   +22.252, E3 +561847.809}
SPL {X  -162.820, Y  +558.919, Z    +0.000, E1   +22.286, E3 +561863.972}
SPL {X  -162.820, Y  +556.169, Z    +0.000, E1   +22.295, E3 +561877.801}
SPL {X  -162.820, Y  +553.294, Z    +0.000, E1   +22.266, E3 +561892.799}
SPL {X  -162.820, Y  +550.136, Z    +0.000, E1   +22.258, E3 +561908.912}
SPL {X  -162.820, Y  +546.694, Z    +0.000, E1   +22.290, E3 +561926.234}
SPL {X  -162.820, Y  +543.558, Z    +0.000, E1   +22.285, E3 +561942.097}
SPL {X  -162.820, Y  +541.633, Z    +0.000, E1   +22.257, E3 +561952.025}
SPL {X  -162.820, Y  +539.116, Z    +0.000, E1   +22.302, E3 +561964.636}
SPL {X  -162.820, Y  +535.523, Z    +0.000, E1   +22.266, E3 +561983.298}
SPL {X  -162.820, Y  +531.757, Z    +0.000, E1   +22.276, E3 +562002.352}
SPL {X  -162.820, Y  +527.980, Z    +0.000, E1   +22.326, E3 +562021.183}
SPL {X  -162.820, Y  +524.599, Z    +0.000, E1   +22.287, E3 +562038.581}
SPL {X  -162.820, Y  +522.011, Z    +0.000, E1   +22.282, E3 +562051.657}
SPL {X  -162.820, Y  +519.457, Z    +0.000, E1   +22.481, E3 +562062.947}
SPL {X  -162.820, Y  +505.859, Z    +0.000, E1   +28.367, E3 +562077.430}
SPL {X  -162.820, Y  +504.131, Z    +0.000, E1   +27.325, E3 +562091.568}
SPL {X  -162.820, Y  +503.215, Z    +0.000, E1   +26.369, E3 +562102.254}
SPL {X  -162.820, Y  +502.502, Z    +0.000, E1   +25.597, E3 +562111.101}
SPL {X  -162.820, Y  +501.672, Z    +0.000, E1   +24.583, E3 +562122.716}
SPL {X  -162.820, Y  +500.515, Z    +0.000, E1   +23.444, E3 +562137.246}
SPL {X  -162.820, Y  +499.633, Z    +0.000, E1   +22.486, E3 +562149.292}
SPL {X  -162.820, Y  +498.303, Z    +0.000, E1   +21.749, E3 +562162.602}
SPL {X  -162.820, Y  +495.897, Z    +0.000, E1   +21.662, E3 +562175.755}
SPL {X  -162.820, Y  +493.717, Z    +0.000, E1   +21.704, E3 +562186.861}
SPL {X  -162.820, Y  +491.396, Z    +0.000, E1   +21.707, E3 +562198.985}
SPL {X  -162.820, Y  +489.485, Z    +0.000, E1   +21.661, E3 +562209.333}
SPL {X  -162.820, Y  +487.723, Z    +0.000, E1   +21.665, E3 +562218.537}
SPL {X  -162.820, Y  +485.661, Z    +0.000, E1   +21.712, E3 +562228.980}
SPL {X  -162.820, Y  +482.775, Z    +0.000, E1   +21.716, E3 +562244.233}
SPL {X  -162.820, Y  +479.894, Z    +0.000, E1   +21.695, E3 +562259.309}
SPL {X  -162.820, Y  +477.685, Z    +0.000, E1   +21.656, E3 +562271.246}
SPL {X  -162.820, Y  +475.419, Z    +0.000, E1   +21.711, E3 +562282.599}
SPL {X  -162.820, Y  +473.301, Z    +0.000, E1   +21.712, E3 +562293.696}
SPL {X  -162.820, Y  +470.965, Z    +0.000, E1   +21.700, E3 +562306.041}
SPL {X  -162.820, Y  +469.036, Z    +0.000, E1   +21.695, E3 +562316.085}
SPL {X  -162.820, Y  +467.138, Z    +0.000, E1   +21.678, E3 +562326.256}
SPL {X  -162.820, Y  +465.011, Z    +0.000, E1   +21.692, E3 +562337.239}
SPL {X  -162.820, Y  +462.669, Z    +0.000, E1   +21.752, E3 +562349.019}
SPL {X  -162.820, Y  +460.725, Z    +0.000, E1   +21.689, E3 +562359.633}
SPL {X  -162.820, Y  +458.666, Z    +0.000, E1   +21.695, E3 +562370.444}
SPL {X  -162.820, Y  +456.431, Z    +0.000, E1   +21.708, E3 +562381.973}
SPL {X  -162.820, Y  +454.628, Z    +0.000, E1   +21.674, E3 +562391.691}
SPL {X  -162.820, Y  +452.690, Z    +0.000, E1   +21.773, E3 +562400.965}
SPL {X  -162.820, Y  +450.610, Z    +0.000, E1   +21.698, E3 +562412.564}
SPL {X  -162.820, Y  +448.170, Z    +0.000, E1   +21.667, E3 +562425.585}
SPL {X  -162.820, Y  +446.246, Z    +0.000, E1   +21.696, E3 +562435.403}
SPL {X  -162.820, Y  +443.784, Z    +0.000, E1   +21.713, E3 +562448.189}
SPL {X  -162.820, Y  +440.567, Z    +0.000, E1   +21.731, E3 +562465.029}
SPL {X  -162.820, Y  +437.628, Z    +0.000, E1   +21.678, E3 +562480.693}
SPL {X  -162.820, Y  +435.262, Z    +0.000, E1   +21.727, E3 +562492.628}
SPL {X  -162.820, Y  +433.510, Z    +0.000, E1   +21.692, E3 +562502.042}
SPL {X  -162.820, Y  +431.492, Z    +0.000, E1   +21.686, E3 +562512.738}
SPL {X  -162.820, Y  +429.074, Z    +0.000, E1   +21.710, E3 +562525.190}
SPL {X  -162.820, Y  +427.020, Z    +0.000, E1   +21.674, E3 +562536.191}
SPL {X  -162.820, Y  +424.525, Z    +0.000, E1   +21.712, E3 +562549.104}
SPL {X  -162.820, Y  +421.144, Z    +0.000, E1   +21.719, E3 +562566.771}
SPL {X  -162.820, Y  +418.116, Z    +0.000, E1   +21.761, E3 +562582.102}
SPL {X  -162.820, Y  +416.127, Z    +0.000, E1   +21.715, E3 +562592.808}
SPL {X  -162.820, Y  +414.361, Z    +0.000, E1   +21.613, E3 +562602.995}
SPL {X  -162.820, Y  +412.134, Z    +0.000, E1   +21.697, E3 +562613.939}
SPL {X  -162.820, Y  +409.248, Z    +0.000, E1   +21.741, E3 +562628.875}
SPL {X  -162.820, Y  +406.238, Z    +0.000, E1   +21.697, E3 +562644.843}
SPL {X  -162.820, Y  +404.001, Z    +0.000, E1   +21.723, E3 +562656.272}
SPL {X  -162.820, Y  +402.223, Z    +0.000, E1   +21.697, E3 +562665.757}
SPL {X  -162.820, Y  +400.348, Z    +0.000, E1   +21.713, E3 +562675.483}
SPL {X  -162.820, Y  +398.298, Z    +0.000, E1   +21.721, E3 +562686.099}
SPL {X  -162.820, Y  +396.371, Z    +0.000, E1   +21.713, E3 +562696.281}
SPL {X  -162.820, Y  +394.508, Z    +0.000, E1   +21.616, E3 +562706.836}
SPL {X  -162.820, Y  +392.435, Z    +0.000, E1   +21.681, E3 +562717.190}
SPL {X  -162.820, Y  +389.390, Z    +0.000, E1   +21.742, E3 +562732.796}
SPL {X  -162.820, Y  +386.818, Z    +0.000, E1   +21.679, E3 +562746.555}
SPL {X  -162.820, Y  +384.697, Z    +0.000, E1   +21.693, E3 +562757.625}
SPL {X  -162.820, Y  +382.288, Z    +0.000, E1   +21.742, E3 +562769.749}
SPL {X  -162.817, Y  +379.520, Z    +0.000, E1   +21.723, E3 +562784.586}
SPL {X  -162.776, Y  +376.710, Z    +0.000, E1   +21.698, E3 +562799.326}
SPL {X  -162.707, Y  +374.438, Z    +0.000, E1   +21.688, E3 +562811.329}
SPL {X  -162.607, Y  +372.171, Z    +0.000, E1   +21.692, E3 +562823.129}
SPL {X  -162.494, Y  +370.197, Z    +0.000, E1   +21.655, E3 +562833.755}
SPL {X  -162.349, Y  +368.131, Z    +0.000, E1   +21.624, E3 +562844.873}
SPL {X  -162.161, Y  +365.866, Z    +0.000, E1   +21.642, E3 +562856.559}
SPL {X  -161.651, Y  +361.024, Z    +0.000, E1   +22.970, E3 +562869.982}
SPL {X  -160.281, Y  +351.857, Z    +0.000, E1   +24.243, E3 +562905.321}
ENDSPLINE

SPLINE
SPL {X  -161.833, Y  +362.603, Z    +0.000, E1   +17.021, E3 +562920.017}
ENDSPLINE

SPLINE
SPL {X  -160.786, Y  +354.842, Z    +0.000, E1   +19.274, E3 +562952.172}
ENDSPLINE

SPLINE
SPL {X  -162.485, Y  +370.062, Z    +0.000, E1   +10.606, E3 +562958.550}
SPL {X  -162.818, Y  +379.636, Z    +0.000, E1    +5.115, E3 +562947.899}
SPL {X  -162.820, Y  +386.976, Z    +0.000, E1    +0.144, E3 +562946.998}
SPL {X  -162.820, Y  +391.982, Z    +0.000, E1    -3.443, E3 +562953.763}
SPL {X  -162.820, Y  +399.630, Z    +0.000, E1    -9.426, E3 +562956.271}
SPL {X  -162.820, Y  +408.127, Z    +0.000, E1   -18.417, E3 +562942.559}
SPL {X  -162.820, Y  +420.083, Z    +0.000, E1   -24.325, E3 +562963.035}
SPL {X  -162.820, Y  +428.527, Z    +0.000, E1   -26.988, E3 +562980.327}
SPL {X  -162.820, Y  +431.336, Z    +0.000, E1   -24.162, E3 +563010.537}
SPL {X  -162.820, Y  +432.048, Z    +0.000, E1   -22.832, E3 +563025.041}
SPL {X  -162.820, Y  +434.888, Z    +0.000, E1   -22.823, E3 +563038.990}
SPL {X  -162.820, Y  +436.834, Z    +0.000, E1   -22.779, E3 +563048.950}
SPL {X  -162.820, Y  +438.868, Z    +0.000, E1   -22.837, E3 +563058.604}
SPL {X  -162.820, Y  +441.351, Z    +0.000, E1   -22.805, E3 +563071.179}
SPL {X  -162.820, Y  +443.809, Z    +0.000, E1   -22.804, E3 +563083.345}
SPL {X  -162.820, Y  +446.105, Z    +0.000, E1   -22.815, E3 +563094.587}
SPL {X  -162.820, Y  +447.974, Z    +0.000, E1   -22.856, E3 +563103.490}
SPL {X  -162.820, Y  +449.911, Z    +0.000, E1   -22.774, E3 +563113.765}
SPL {X  -162.820, Y  +451.861, Z    +0.000, E1   -22.750, E3 +563123.613}
SPL {X  -162.820, Y  +454.167, Z    +0.000, E1   -22.842, E3 +563134.342}
SPL {X  -162.820, Y  +456.529, Z    +0.000, E1   -22.855, E3 +563145.870}
SPL {X  -162.820, Y  +458.725, Z    +0.000, E1   -22.793, E3 +563157.275}
SPL {X  -162.820, Y  +461.700, Z    +0.000, E1   -22.822, E3 +563171.897}
SPL {X  -162.820, Y  +464.633, Z    +0.000, E1   -22.813, E3 +563186.394}
SPL {X  -162.820, Y  +466.699, Z    +0.000, E1   -22.824, E3 +563196.440}
SPL {X  -162.820, Y  +468.655, Z    +0.000, E1   -22.858, E3 +563205.884}
SPL {X  -162.820, Y  +470.892, Z    +0.000, E1   -22.837, E3 +563217.123}
SPL {X  -162.820, Y  +473.485, Z    +0.000, E1   -22.806, E3 +563230.321}
SPL {X  -162.820, Y  +476.589, Z    +0.000, E1   -22.788, E3 +563245.843}
SPL {X  -162.820, Y  +478.914, Z    +0.000, E1   -22.821, E3 +563256.941}
SPL {X  -162.820, Y  +481.034, Z    +0.000, E1   -22.831, E3 +563267.463}
SPL {X  -162.820, Y  +484.256, Z    +0.000, E1   -22.840, E3 +563283.482}
SPL {X  -162.820, Y  +487.014, Z    +0.000, E1   -22.789, E3 +563297.349}
SPL {X  -162.820, Y  +489.750, Z    +0.000, E1   -22.832, E3 +563310.723}
SPL {X  -162.820, Y  +493.233, Z    +0.000, E1   -22.844, E3 +563327.860}
SPL {X  -162.820, Y  +496.150, Z    +0.000, E1   -22.796, E3 +563342.579}
SPL {X  -162.820, Y  +498.661, Z    +0.000, E1   -22.828, E3 +563354.760}
SPL {X  -162.820, Y  +501.761, Z    +0.000, E1   -22.820, E3 +563370.329}
SPL {X  -162.820, Y  +505.323, Z    +0.000, E1   -22.838, E3 +563387.776}
SPL {X  -162.820, Y  +507.875, Z    +0.000, E1   -22.849, E3 +563400.143}
SPL {X  -162.820, Y  +510.068, Z    +0.000, E1   -22.761, E3 +563411.836}
SPL {X  -162.820, Y  +512.359, Z    +0.000, E1   -22.823, E3 +563422.568}
SPL {X  -162.820, Y  +514.562, Z    +0.000, E1   -22.806, E3 +563433.754}
SPL {X  -162.820, Y  +517.952, Z    +0.000, E1   -22.864, E3 +563450.152}
SPL {X  -162.820, Y  +520.641, Z    +0.000, E1   -22.790, E3 +563463.870}
SPL {X  -162.820, Y  +522.740, Z    +0.000, E1   -22.811, E3 +563474.113}
SPL {X  -162.820, Y  +524.628, Z    +0.000, E1   -22.846, E3 +563483.108}
SPL {X  -162.820, Y  +526.661, Z    +0.000, E1   -22.801, E3 +563493.663}
SPL {X  -162.820, Y  +529.662, Z    +0.000, E1   -22.810, E3 +563508.514}
SPL {X  -162.820, Y  +532.614, Z    +0.000, E1   -22.828, E3 +563522.920}
SPL {X  -162.820, Y  +534.838, Z    +0.000, E1   -22.864, E3 +563533.549}
SPL {X  -162.820, Y  +536.882, Z    +0.000, E1   -22.782, E3 +563544.404}
SPL {X  -162.820, Y  +539.194, Z    +0.000, E1   -22.826, E3 +563555.452}
SPL {X  -162.820, Y  +541.555, Z    +0.000, E1   -22.817, E3 +563567.267}
SPL {X  -162.820, Y  +543.728, Z    +0.000, E1   -22.799, E3 +563578.124}
SPL {X  -162.820, Y  +545.925, Z    +0.000, E1   -22.803, E3 +563588.994}
SPL {X  -162.820, Y  +549.071, Z    +0.000, E1   -22.836, E3 +563604.522}
SPL {X  -162.820, Y  +553.089, Z    +0.000, E1   -22.838, E3 +563624.422}
SPL {X  -162.820, Y  +556.430, Z    +0.000, E1   -22.821, E3 +563640.923}
SPL {X  -162.820, Y  +558.974, Z    +0.000, E1   -22.806, E3 +563653.623}
SPL {X  -162.820, Y  +562.171, Z    +0.000, E1   -22.845, E3 +563669.321}
SPL {X  -162.820, Y  +565.170, Z    +0.000, E1   -22.801, E3 +563684.334}
SPL {X  -162.820, Y  +567.308, Z    +0.000, E1   -22.750, E3 +563695.350}
SPL {X  -162.820, Y  +570.378, Z    +0.000, E1   -22.843, E3 +563709.974}
SPL {X  -162.820, Y  +573.634, Z    +0.000, E1   -22.827, E3 +563726.118}
SPL {X  -162.820, Y  +576.228, Z    +0.000, E1   -22.814, E3 +563739.014}
SPL {X  -162.820, Y  +578.553, Z    +0.000, E1   -22.801, E3 +563750.630}
SPL {X  -162.820, Y  +581.064, Z    +0.000, E1   -22.823, E3 +563762.915}
SPL {X  -162.820, Y  +583.435, Z    +0.000, E1   -22.808, E3 +563774.736}
SPL {X  -162.820, Y  +585.410, Z    +0.000, E1   -22.764, E3 +563784.872}
SPL {X  -162.820, Y  +587.676, Z    +0.000, E1   -22.853, E3 +563795.387}
SPL {X  -162.820, Y  +590.707, Z    +0.000, E1   -22.855, E3 +563810.537}
SPL {X  -162.820, Y  +593.650, Z    +0.000, E1   -22.810, E3 +563825.297}
SPL {X  -162.820, Y  +595.830, Z    +0.000, E1   -22.828, E3 +563835.913}
SPL {X  -162.820, Y  +598.094, Z    +0.000, E1   -22.843, E3 +563847.026}
SPL {X  -162.820, Y  +600.420, Z    +0.000, E1   -22.826, E3 +563858.657}
SPL {X  -162.820, Y  +602.573, Z    +0.000, E1   -22.830, E3 +563869.243}
SPL {X  -162.820, Y  +604.828, Z    +0.000, E1   -22.784, E3 +563880.881}
SPL {X  -162.820, Y  +608.133, Z    +0.000, E1   -22.831, E3 +563896.999}
SPL {X  -162.820, Y  +611.103, Z    +0.000, E1   -22.785, E3 +563911.924}
SPL {X  -162.820, Y  +613.294, Z    +0.000, E1   -22.780, E3 +563922.798}
SPL {X  -162.820, Y  +615.356, Z    +0.000, E1   -22.799, E3 +563932.855}
SPL {X  -162.820, Y  +617.439, Z    +0.000, E1   -22.808, E3 +563943.113}
SPL {X  -162.820, Y  +619.665, Z    +0.000, E1   -22.817, E3 +563954.081}
SPL {X  -162.820, Y  +621.733, Z    +0.000, E1   -22.759, E3 +563964.805}
SPL {X  -162.820, Y  +624.076, Z    +0.000, E1   -22.774, E3 +563976.310}
SPL {X  -162.820, Y  +626.527, Z    +0.000, E1   -22.768, E3 +563988.553}
SPL {X  -162.820, Y  +629.758, Z    +0.000, E1   -22.800, E3 +564004.482}
SPL {X  -162.820, Y  +632.572, Z    +0.000, E1   -22.785, E3 +564018.331}
SPL {X  -162.820, Y  +634.507, Z    +0.000, E1   -22.784, E3 +564027.970}
SPL {X  -162.820, Y  +636.863, Z    +0.000, E1   -22.760, E3 +564039.892}
SPL {X  -162.820, Y  +639.254, Z    +0.000, E1   -22.767, E3 +564051.675}
SPL {X  -162.820, Y  +641.888, Z    +0.000, E1   -22.790, E3 +564064.622}
SPL {X  -162.820, Y  +644.915, Z    +0.000, E1   -22.818, E3 +564079.397}
SPL {X  -162.820, Y  +647.561, Z    +0.000, E1   -22.705, E3 +564093.439}
SPL {X  -162.820, Y  +649.758, Z    +0.000, E1   -22.780, E3 +564103.629}
SPL {X  -162.820, Y  +651.708, Z    +0.000, E1   -22.810, E3 +564113.124}
SPL {X  -162.820, Y  +653.898, Z    +0.000, E1   -22.796, E3 +564124.044}
SPL {X  -162.820, Y  +656.161, Z    +0.000, E1   -22.812, E3 +564135.166}
SPL {X  -162.820, Y  +658.384, Z    +0.000, E1   -22.822, E3 +564146.032}
SPL {X  -162.820, Y  +660.215, Z    +0.000, E1   -22.649, E3 +564156.623}
SPL {X  -162.820, Y  +662.823, Z    +0.000, E1   -22.799, E3 +564168.331}
SPL {X  -162.820, Y  +665.862, Z    +0.000, E1   -22.864, E3 +564183.030}
SPL {X  -162.820, Y  +668.960, Z    +0.000, E1   -22.773, E3 +564198.981}
SPL {X  -162.820, Y  +671.605, Z    +0.000, E1   -22.777, E3 +564212.055}
SPL {X  -162.817, Y  +674.515, Z    +0.000, E1   -22.816, E3 +564226.252}
SPL {X  -162.773, Y  +677.428, Z    +0.000, E1   -22.762, E3 +564241.060}
SPL {X  -162.691, Y  +679.987, Z    +0.000, E1   -22.794, E3 +564253.473}
SPL {X  -162.559, Y  +682.717, Z    +0.000, E1   -22.726, E3 +564267.656}
SPL {X  -162.404, Y  +685.137, Z    +0.000, E1   -22.766, E3 +564279.179}
SPL {X  -162.229, Y  +687.364, Z    +0.000, E1   -22.685, E3 +564291.047}
SPL {X  -161.938, Y  +690.422, Z    +0.000, E1   -22.769, E3 +564305.453}
SPL {X  -161.065, Y  +697.344, Z    +0.000, E1   -25.698, E3 +564314.573}
SPL {X  -158.553, Y  +710.529, Z    +0.000, E1   -30.890, E3 +564328.469}
ENDSPLINE

SPLINE
SPL {X  -161.215, Y  +696.305, Z    +0.000, E1   -20.575, E3 +564355.050}
SPL {X  -161.691, Y  +692.643, Z    +0.000, E1   -17.369, E3 +564371.238}
SPL {X  -162.534, Y  +683.153, Z    +0.000, E1   -10.475, E3 +564396.705}
SPL {X  -162.820, Y  +670.105, Z    +0.000, E1    -2.484, E3 +564389.352}
SPL {X  -162.820, Y  +665.819, Z    +0.000, E1    +0.492, E3 +564391.649}
SPL {X  -162.820, Y  +661.883, Z    +0.000, E1    +3.373, E3 +564396.125}
SPL {X  -162.820, Y  +655.163, Z    +0.000, E1    +8.702, E3 +564395.724}
SPL {X  -162.820, Y  +634.515, Z    +0.000, E1   +26.439, E3 +564388.137}
ENDSPLINE

SPLINE
SPL {X  -162.820, Y  +638.080, Z    +0.000, E1   +18.858, E3 +564418.101}
ENDSPLINE

SPLINE
SPL {X  -162.820, Y  +623.278, Z    +0.000, E1   +28.723, E3 +564419.672}
SPL {X  -162.820, Y  +611.829, Z    +0.000, E1   +31.229, E3 +564443.324}
ENDSPLINE

SPLINE
SPL {X  -162.820, Y  +623.595, Z    +0.000, E1   +22.712, E3 +564458.245}
ENDSPLINE

SPLINE
SPL {X  -162.820, Y  +621.304, Z    +0.000, E1   +22.259, E3 +564473.403}
SPL {X  -162.820, Y  +618.758, Z    +0.000, E1   +22.239, E3 +564486.554}
SPL {X  -162.820, Y  +616.062, Z    +0.000, E1   +22.275, E3 +564499.974}
SPL {X  -162.820, Y  +613.536, Z    +0.000, E1   +22.242, E3 +564513.096}
SPL {X  -162.820, Y  +611.128, Z    +0.000, E1   +22.252, E3 +564525.267}
SPL {X  -162.820, Y  +608.428, Z    +0.000, E1   +22.255, E3 +564539.050}
SPL {X  -162.820, Y  +605.178, Z    +0.000, E1   +22.267, E3 +564555.582}
SPL {X  -162.820, Y  +602.350, Z    +0.000, E1   +22.224, E3 +564570.199}
SPL {X  -162.820, Y  +599.842, Z    +0.000, E1   +22.298, E3 +564582.351}
SPL {X  -162.820, Y  +597.194, Z    +0.000, E1   +22.253, E3 +564596.272}
SPL {X  -162.820, Y  +594.779, Z    +0.000, E1   +22.284, E3 +564608.176}
SPL {X  -162.820, Y  +593.320, Z    +0.000, E1   +22.199, E3 +564616.279}
SPL {X  -162.820, Y  +591.031, Z    +0.000, E1   +22.283, E3 +564627.370}
SPL {X  -162.820, Y  +588.026, Z    +0.000, E1   +22.301, E3 +564642.497}
SPL {X  -162.820, Y  +585.899, Z    +0.000, E1   +22.286, E3 +564653.299}
SPL {X  -162.820, Y  +583.204, Z    +0.000, E1   +22.278, E3 +564667.322}
SPL {X  -162.820, Y  +579.691, Z    +0.000, E1   +22.312, E3 +564684.810}
SPL {X  -162.820, Y  +577.460, Z    +0.000, E1   +22.218, E3 +564696.797}
SPL {X  -162.820, Y  +575.394, Z    +0.000, E1   +22.240, E3 +564707.222}
SPL {X  -162.820, Y  +572.645, Z    +0.000, E1   +22.246, E3 +564721.220}
SPL {X  -162.820, Y  +570.282, Z    +0.000, E1   +22.231, E3 +564733.270}
SPL {X  -162.820, Y  +567.961, Z    +0.000, E1   +22.247, E3 +564745.060}
SPL {X  -162.820, Y  +564.506, Z    +0.000, E1   +22.298, E3 +564762.374}
SPL {X  -162.820, Y  +561.620, Z    +0.000, E1   +22.191, E3 +564777.755}
SPL {X  -162.820, Y  +559.515, Z    +0.000, E1   +22.273, E3 +564787.757}
SPL {X  -162.820, Y  +556.723, Z    +0.000, E1   +22.309, E3 +564801.840}
SPL {X  -162.820, Y  +554.378, Z    +0.000, E1   +22.288, E3 +564813.686}
SPL {X  -162.820, Y  +552.787, Z    +0.000, E1   +22.213, E3 +564822.508}
SPL {X  -162.820, Y  +550.871, Z    +0.000, E1   +22.229, E3 +564832.102}
SPL {X  -162.820, Y  +548.168, Z    +0.000, E1   +22.298, E3 +564845.438}
SPL {X  -162.820, Y  +545.860, Z    +0.000, E1   +22.216, E3 +564857.696}
SPL {X  -162.820, Y  +543.558, Z    +0.000, E1   +22.285, E3 +564868.926}
SPL {X  -162.820, Y  +540.968, Z    +0.000, E1   +22.274, E3 +564882.199}
SPL {X  -162.820, Y  +538.512, Z    +0.000, E1   +22.287, E3 +564894.511}
SPL {X  -162.820, Y  +535.523, Z    +0.000, E1   +22.266, E3 +564910.127}
SPL {X  -162.820, Y  +531.757, Z    +0.000, E1   +22.276, E3 +564929.181}
SPL {X  -162.820, Y  +527.980, Z    +0.000, E1   +22.326, E3 +564948.012}
SPL {X  -162.820, Y  +524.599, Z    +0.000, E1   +22.287, E3 +564965.410}
SPL {X  -162.820, Y  +522.011, Z    +0.000, E1   +22.282, E3 +564978.487}
SPL {X  -162.820, Y  +519.457, Z    +0.000, E1   +22.481, E3 +564989.776}
SPL {X  -162.820, Y  +505.859, Z    +0.000, E1   +28.367, E3 +565004.259}
SPL {X  -162.820, Y  +504.131, Z    +0.000, E1   +27.325, E3 +565018.397}
SPL {X  -162.820, Y  +502.813, Z    +0.000, E1   +26.013, E3 +565033.774}
SPL {X  -162.820, Y  +502.016, Z    +0.000, E1   +24.802, E3 +565046.116}
SPL {X  -162.820, Y  +501.060, Z    +0.000, E1   +24.081, E3 +565056.306}
SPL {X  -162.820, Y  +499.934, Z    +0.000, E1   +22.814, E3 +565072.175}
SPL {X  -162.820, Y  +498.303, Z    +0.000, E1   +21.749, E3 +565089.431}
SPL {X  -162.820, Y  +495.897, Z    +0.000, E1   +21.662, E3 +565102.584}
SPL {X  -162.820, Y  +493.717, Z    +0.000, E1   +21.704, E3 +565113.691}
SPL {X  -162.820, Y  +491.396, Z    +0.000, E1   +21.707, E3 +565125.815}
SPL {X  -162.820, Y  +489.485, Z    +0.000, E1   +21.661, E3 +565136.163}
SPL {X  -162.820, Y  +487.723, Z    +0.000, E1   +21.665, E3 +565145.366}
SPL {X  -162.820, Y  +485.661, Z    +0.000, E1   +21.712, E3 +565155.809}
SPL {X  -162.820, Y  +482.775, Z    +0.000, E1   +21.716, E3 +565171.062}
SPL {X  -162.820, Y  +479.894, Z    +0.000, E1   +21.695, E3 +565186.138}
SPL {X  -162.820, Y  +477.685, Z    +0.000, E1   +21.656, E3 +565198.076}
SPL {X  -162.820, Y  +475.419, Z    +0.000, E1   +21.711, E3 +565209.428}
SPL {X  -162.820, Y  +473.301, Z    +0.000, E1   +21.712, E3 +565220.525}
SPL {X  -162.820, Y  +470.965, Z    +0.000, E1   +21.700, E3 +565232.870}
SPL {X  -162.820, Y  +469.036, Z    +0.000, E1   +21.695, E3 +565242.914}
SPL {X  -162.820, Y  +467.138, Z    +0.000, E1   +21.678, E3 +565253.086}
SPL {X  -162.820, Y  +465.011, Z    +0.000, E1   +21.692, E3 +565264.068}
SPL {X  -162.820, Y  +462.669, Z    +0.000, E1   +21.752, E3 +565275.849}
SPL {X  -162.820, Y  +460.725, Z    +0.000, E1   +21.689, E3 +565286.462}
SPL {X  -162.820, Y  +458.666, Z    +0.000, E1   +21.695, E3 +565297.274}
SPL {X  -162.820, Y  +456.431, Z    +0.000, E1   +21.708, E3 +565308.802}
SPL {X  -162.820, Y  +454.628, Z    +0.000, E1   +21.674, E3 +565318.521}
SPL {X  -162.820, Y  +452.690, Z    +0.000, E1   +21.773, E3 +565327.795}
SPL {X  -162.820, Y  +450.610, Z    +0.000, E1   +21.698, E3 +565339.393}
SPL {X  -162.820, Y  +448.170, Z    +0.000, E1   +21.667, E3 +565352.414}
SPL {X  -162.820, Y  +446.246, Z    +0.000, E1   +21.696, E3 +565362.232}
SPL {X  -162.820, Y  +443.784, Z    +0.000, E1   +21.713, E3 +565375.018}
SPL {X  -162.820, Y  +440.567, Z    +0.000, E1   +21.731, E3 +565391.858}
SPL {X  -162.820, Y  +437.628, Z    +0.000, E1   +21.678, E3 +565407.522}
SPL {X  -162.820, Y  +435.262, Z    +0.000, E1   +21.727, E3 +565419.458}
SPL {X  -162.820, Y  +433.510, Z    +0.000, E1   +21.692, E3 +565428.872}
SPL {X  -162.820, Y  +431.492, Z    +0.000, E1   +21.686, E3 +565439.567}
SPL {X  -162.820, Y  +429.074, Z    +0.000, E1   +21.710, E3 +565452.019}
SPL {X  -162.820, Y  +427.020, Z    +0.000, E1   +21.674, E3 +565463.020}
SPL {X  -162.820, Y  +425.215, Z    +0.000, E1   +21.693, E3 +565472.323}
SPL {X  -162.820, Y  +422.986, Z    +0.000, E1   +21.685, E3 +565484.134}
SPL {X  -162.820, Y  +420.528, Z    +0.000, E1   +21.706, E3 +565496.784}
SPL {X  -162.820, Y  +418.116, Z    +0.000, E1   +21.761, E3 +565508.932}
SPL {X  -162.820, Y  +416.127, Z    +0.000, E1   +21.715, E3 +565519.637}
SPL {X  -162.820, Y  +414.361, Z    +0.000, E1   +21.613, E3 +565529.824}
SPL {X  -162.820, Y  +411.450, Z    +0.000, E1   +21.710, E3 +565544.397}
SPL {X  -162.820, Y  +408.590, Z    +0.000, E1   +21.735, E3 +565559.023}
SPL {X  -162.820, Y  +406.238, Z    +0.000, E1   +21.697, E3 +565571.672}
SPL {X  -162.820, Y  +403.166, Z    +0.000, E1   +21.746, E3 +565587.478}
SPL {X  -162.820, Y  +400.348, Z    +0.000, E1   +21.713, E3 +565602.313}
SPL {X  -162.820, Y  +398.298, Z    +0.000, E1   +21.721, E3 +565612.928}
SPL {X  -162.820, Y  +396.371, Z    +0.000, E1   +21.713, E3 +565623.110}
SPL {X  -162.820, Y  +394.508, Z    +0.000, E1   +21.616, E3 +565633.665}
SPL {X  -162.820, Y  +391.777, Z    +0.000, E1   +21.714, E3 +565647.325}
SPL {X  -162.820, Y  +388.822, Z    +0.000, E1   +21.717, E3 +565662.645}
SPL {X  -162.820, Y  +386.818, Z    +0.000, E1   +21.679, E3 +565673.384}
SPL {X  -162.820, Y  +384.697, Z    +0.000, E1   +21.693, E3 +565684.455}
SPL {X  -162.820, Y  +382.288, Z    +0.000, E1   +21.742, E3 +565696.578}
SPL {X  -162.817, Y  +379.520, Z    +0.000, E1   +21.723, E3 +565711.416}
SPL {X  -162.776, Y  +376.710, Z    +0.000, E1   +21.698, E3 +565726.155}
SPL {X  -162.707, Y  +374.438, Z    +0.000, E1   +21.688, E3 +565738.159}
SPL {X  -162.607, Y  +372.171, Z    +0.000, E1   +21.692, E3 +565749.958}
SPL {X  -162.494, Y  +370.197, Z    +0.000, E1   +21.655, E3 +565760.585}
SPL {X  -162.349, Y  +368.131, Z    +0.000, E1   +21.624, E3 +565771.703}
SPL {X  -162.161, Y  +365.866, Z    +0.000, E1   +21.642, E3 +565783.388}
SPL {X  -161.651, Y  +361.024, Z    +0.000, E1   +22.970, E3 +565796.811}
SPL {X  -160.281, Y  +351.857, Z    +0.000, E1   +24.243, E3 +565832.150}
ENDSPLINE

SPLINE
SPL {X  -161.833, Y  +362.603, Z    +0.000, E1   +17.021, E3 +565846.846}
ENDSPLINE

SPLINE
SPL {X  -160.786, Y  +354.842, Z    +0.000, E1   +19.274, E3 +565879.002}
ENDSPLINE

